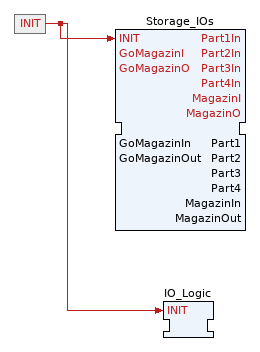
      [picture p72: application VDMA_Station1_EmulatorApp_SingleDevice.Storage]
      SUBAPPLICATION Storage_IOs
        EVENT_INPUT
          INIT;
          GoMagazinI;
          GoMagazinO;
        END_EVENT
        EVENT_OUTPUT
          Part1In;
          Part2In;
          Part3In;
          Part4In;
          MagazinI;
          MagazinO;
        END_EVENT
        VAR_INPUT
          GoMagazinIn : BOOL;
          GoMagazinOut : BOOL;
        END_VAR
        VAR_OUTPUT
          Part1 : BOOL;
          Part2 : BOOL;
          Part3 : BOOL;
          Part4 : BOOL;
          MagazinIn : BOOL;
          MagazinOut : BOOL;
        END_VAR
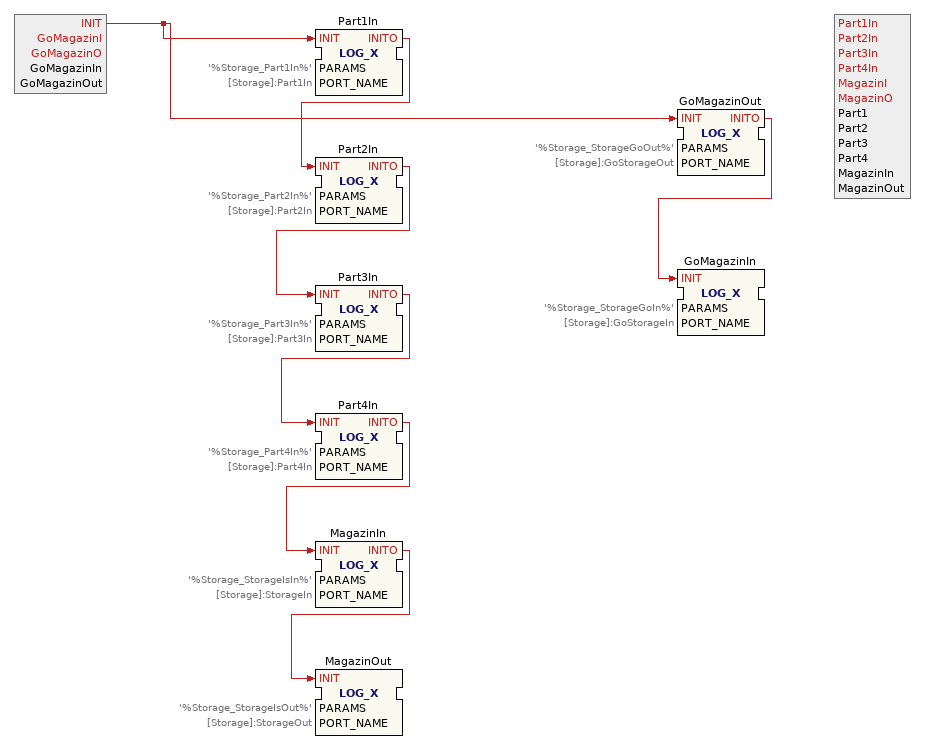
        FBS
          GoMagazinIn : LOG_X(PARAMS := '%Storage_StorageGoIn%', PORT_NAME := [Storage]:GoStorageIn);
          GoMagazinOut : LOG_X(PARAMS := '%Storage_StorageGoOut%', PORT_NAME := [Storage]:GoStorageOut);
          MagazinOut : LOG_X(PARAMS := '%Storage_StorageIsOut%', PORT_NAME := [Storage]:StorageOut);
          MagazinIn : LOG_X(PARAMS := '%Storage_StorageIsIn%', PORT_NAME := [Storage]:StorageIn);
          Part4In : LOG_X(PARAMS := '%Storage_Part4In%', PORT_NAME := [Storage]:Part4In);
          Part3In : LOG_X(PARAMS := '%Storage_Part3In%', PORT_NAME := [Storage]:Part3In);
          Part2In : LOG_X(PARAMS := '%Storage_Part2In%', PORT_NAME := [Storage]:Part2In);
          Part1In : LOG_X(PARAMS := '%Storage_Part1In%', PORT_NAME := [Storage]:Part1In);
        END_FBS
        EVENT_CONNECTIONS
          GoMagazinOut.INITO TO GoMagazinIn.INIT;
          MagazinIn.INITO TO MagazinOut.INIT;
          Part4In.INITO TO MagazinIn.INIT;
          Part3In.INITO TO Part4In.INIT;
          Part2In.INITO TO Part3In.INIT;
          Part1In.INITO TO Part2In.INIT;
          INIT TO Part1In.INIT;
          INIT TO GoMagazinOut.INIT;
        END_CONNECTIONS
      END_SUBAPPLICATION
      SUBAPPLICATION IO_Logic
        EVENT_INPUT
          INIT;
        END_EVENT
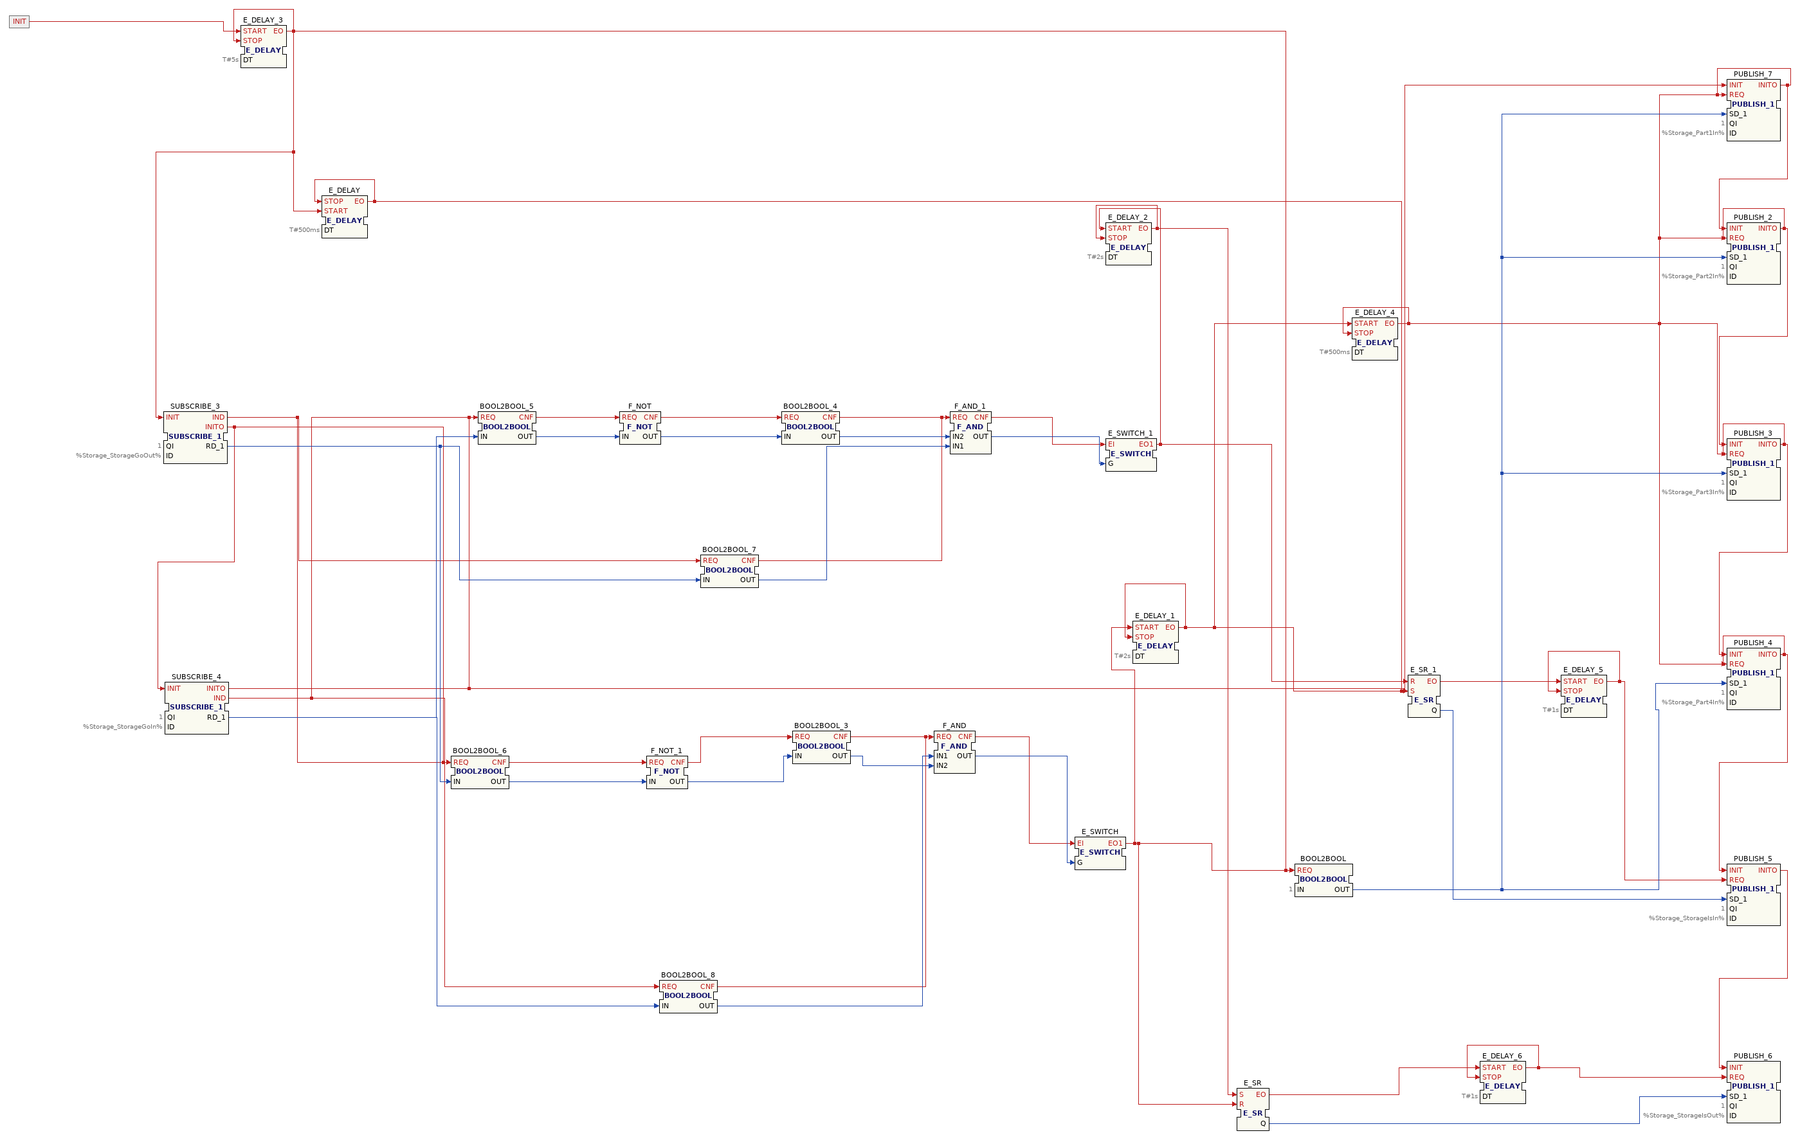
        FBS
          E_SWITCH_1 : E_SWITCH;
          BOOL2BOOL_4 : BOOL2BOOL;
          F_NOT : F_NOT;
          PUBLISH_3 : PUBLISH_1(QI := 1, ID := %Storage_Part3In%);
          BOOL2BOOL_6 : BOOL2BOOL;
          E_SR_1 : E_SR;
          F_NOT_1 : F_NOT;
          PUBLISH_7 : PUBLISH_1(QI := 1, ID := %Storage_Part1In%);
          BOOL2BOOL : BOOL2BOOL(IN := 1);
          BOOL2BOOL_5 : BOOL2BOOL;
          BOOL2BOOL_7 : BOOL2BOOL;
          E_SR : E_SR;
          F_AND_1 : F_AND;
          SUBSCRIBE_4 : SUBSCRIBE_1(QI := 1, ID := %Storage_StorageGoIn%);
          SUBSCRIBE_3 : SUBSCRIBE_1(QI := 1, ID := %Storage_StorageGoOut%);
          PUBLISH_6 : PUBLISH_1(QI := 1, ID := %Storage_StorageIsOut%);
          F_AND : F_AND;
          BOOL2BOOL_3 : BOOL2BOOL;
          PUBLISH_5 : PUBLISH_1(QI := 1, ID := %Storage_StorageIsIn%);
          PUBLISH_4 : PUBLISH_1(QI := 1, ID := %Storage_Part4In%);
          E_DELAY_2 : E_DELAY(DT := T#2s);
          BOOL2BOOL_8 : BOOL2BOOL;
          E_DELAY_1 : E_DELAY(DT := T#2s);
          PUBLISH_2 : PUBLISH_1(QI := 1, ID := %Storage_Part2In%);
          E_SWITCH : E_SWITCH;
          E_DELAY : E_DELAY(DT := T#500ms);
          E_DELAY_3 : E_DELAY(DT := T#5s);
          E_DELAY_4 : E_DELAY(DT := T#500ms);
          E_DELAY_5 : E_DELAY(DT := T#1s);
          E_DELAY_6 : E_DELAY(DT := T#1s);
        END_FBS
        EVENT_CONNECTIONS
          F_AND_1.CNF TO E_SWITCH_1.EI;
          E_SWITCH_1.EO1 TO E_SR_1.R;
          E_SWITCH_1.EO1 TO E_DELAY_2.START;
          F_NOT.CNF TO BOOL2BOOL_4.REQ;
          BOOL2BOOL_4.CNF TO F_AND_1.REQ;
          BOOL2BOOL_5.CNF TO F_NOT.REQ;
          PUBLISH_2.INITO TO PUBLISH_3.INIT;
          PUBLISH_3.INITO TO PUBLISH_3.REQ;
          PUBLISH_3.INITO TO PUBLISH_4.INIT;
          SUBSCRIBE_3.IND TO BOOL2BOOL_6.REQ;
          SUBSCRIBE_3.INITO TO BOOL2BOOL_6.REQ;
          BOOL2BOOL_6.CNF TO F_NOT_1.REQ;
          E_DELAY_1.EO TO E_SR_1.S;
          F_NOT_1.CNF TO BOOL2BOOL_3.REQ;
          SUBSCRIBE_4.INITO TO PUBLISH_7.INIT;
          PUBLISH_7.INITO TO PUBLISH_7.REQ;
          PUBLISH_7.INITO TO PUBLISH_2.INIT;
          E_SWITCH.EO1 TO BOOL2BOOL.REQ;
          SUBSCRIBE_4.IND TO BOOL2BOOL_5.REQ;
          SUBSCRIBE_4.INITO TO BOOL2BOOL_5.REQ;
          SUBSCRIBE_3.IND TO BOOL2BOOL_7.REQ;
          BOOL2BOOL_7.CNF TO F_AND_1.REQ;
          E_DELAY_2.EO TO E_SR.S;
          E_SWITCH.EO1 TO E_SR.R;
          SUBSCRIBE_3.INITO TO SUBSCRIBE_4.INIT;
          SUBSCRIBE_4.IND TO BOOL2BOOL_8.REQ;
          PUBLISH_5.INITO TO PUBLISH_6.INIT;
          BOOL2BOOL_3.CNF TO F_AND.REQ;
          BOOL2BOOL_8.CNF TO F_AND.REQ;
          F_AND.CNF TO E_SWITCH.EI;
          PUBLISH_4.INITO TO PUBLISH_5.INIT;
          PUBLISH_4.INITO TO PUBLISH_4.REQ;
          E_DELAY_2.EO TO E_DELAY_2.STOP;
          E_SWITCH.EO1 TO E_DELAY_1.START;
          E_DELAY_1.EO TO E_DELAY_1.STOP;
          PUBLISH_2.INITO TO PUBLISH_2.REQ;
          E_DELAY.EO TO E_DELAY.STOP;
          E_DELAY.EO TO E_SR_1.S;
          E_DELAY_3.EO TO BOOL2BOOL.REQ;
          E_DELAY_3.EO TO E_DELAY.START;
          E_DELAY_3.EO TO SUBSCRIBE_3.INIT;
          INIT TO E_DELAY_3.START;
          E_DELAY_3.EO TO E_DELAY_3.STOP;
          E_DELAY_4.EO TO PUBLISH_2.REQ;
          E_DELAY_4.EO TO PUBLISH_4.REQ;
          E_DELAY_4.EO TO PUBLISH_7.REQ;
          E_DELAY_4.EO TO PUBLISH_3.REQ;
          E_DELAY_1.EO TO E_DELAY_4.START;
          E_DELAY_4.EO TO E_DELAY_4.STOP;
          E_SR_1.EO TO E_DELAY_5.START;
          E_DELAY_5.EO TO PUBLISH_5.REQ;
          E_DELAY_5.EO TO E_DELAY_5.STOP;
          E_SR.EO TO E_DELAY_6.START;
          E_DELAY_6.EO TO PUBLISH_6.REQ;
          E_DELAY_6.EO TO E_DELAY_6.STOP;
        END_CONNECTIONS
        DATA_CONNECTIONS
          F_AND_1.OUT TO E_SWITCH_1.G;
          F_NOT.OUT TO BOOL2BOOL_4.IN;
          BOOL2BOOL_4.OUT TO F_AND_1.IN2;
          BOOL2BOOL_5.OUT TO F_NOT.IN;
          BOOL2BOOL.OUT TO PUBLISH_3.SD_1;
          SUBSCRIBE_3.RD_1 TO BOOL2BOOL_6.IN;
          BOOL2BOOL_6.OUT TO F_NOT_1.IN;
          F_NOT_1.OUT TO BOOL2BOOL_3.IN;
          BOOL2BOOL.OUT TO PUBLISH_7.SD_1;
          BOOL2BOOL.OUT TO PUBLISH_4.SD_1;
          BOOL2BOOL.OUT TO PUBLISH_2.SD_1;
          SUBSCRIBE_4.RD_1 TO BOOL2BOOL_5.IN;
          SUBSCRIBE_3.RD_1 TO BOOL2BOOL_7.IN;
          BOOL2BOOL_7.OUT TO F_AND_1.IN1;
          E_SR.Q TO PUBLISH_6.SD_1;
          SUBSCRIBE_4.RD_1 TO BOOL2BOOL_8.IN;
          BOOL2BOOL_8.OUT TO F_AND.IN1;
          BOOL2BOOL_3.OUT TO F_AND.IN2;
          F_AND.OUT TO E_SWITCH.G;
          E_SR_1.Q TO PUBLISH_5.SD_1;
        END_CONNECTIONS
      END_SUBAPPLICATION
      EVENT_CONNECTIONS
        INIT TO Storage_IOs.INIT;
        INIT TO IO_Logic.INIT;
      END_CONNECTIONS
    END_SUBAPPLICATION
    SUBAPPLICATION Gripper1
      EVENT_INPUT
        INIT;
      END_EVENT
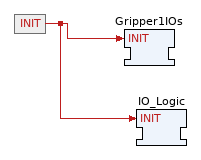
      SUBAPPLICATION Gripper1IOs
        EVENT_INPUT
          INIT;
        END_EVENT
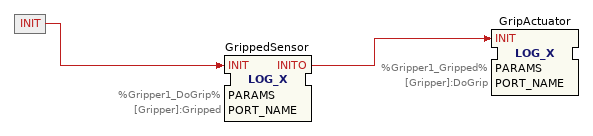
        FBS
          GripActuator : LOG_X(PARAMS := %Gripper1_Gripped%, PORT_NAME := [Gripper]:DoGrip);
          GrippedSensor : LOG_X(PARAMS := %Gripper1_DoGrip%, PORT_NAME := [Gripper]:Gripped);
        END_FBS
        EVENT_CONNECTIONS
          INIT TO GrippedSensor.INIT;
          GrippedSensor.INITO TO GripActuator.INIT;
        END_CONNECTIONS
      END_SUBAPPLICATION
      SUBAPPLICATION IO_Logic
        EVENT_INPUT
          INIT;
        END_EVENT
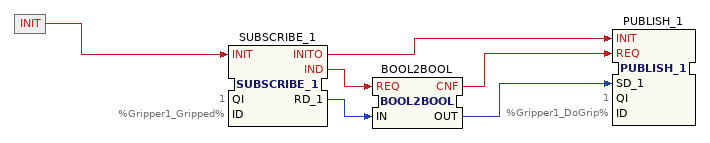
        FBS
          SUBSCRIBE_1 : SUBSCRIBE_1(QI := 1, ID := %Gripper1_Gripped%);
          BOOL2BOOL : BOOL2BOOL;
          PUBLISH_1 : PUBLISH_1(QI := 1, ID := %Gripper1_DoGrip%);
        END_FBS
        EVENT_CONNECTIONS
          SUBSCRIBE_1.INITO TO PUBLISH_1.INIT;
          SUBSCRIBE_1.IND TO BOOL2BOOL.REQ;
          BOOL2BOOL.CNF TO PUBLISH_1.REQ;
          INIT TO SUBSCRIBE_1.INIT;
        END_CONNECTIONS
        DATA_CONNECTIONS
          SUBSCRIBE_1.RD_1 TO BOOL2BOOL.IN;
          BOOL2BOOL.OUT TO PUBLISH_1.SD_1;
        END_CONNECTIONS
      END_SUBAPPLICATION
      EVENT_CONNECTIONS
        INIT TO IO_Logic.INIT;
        INIT TO Gripper1IOs.INIT;
      END_CONNECTIONS
    END_SUBAPPLICATION
    SUBAPPLICATION Gripper2
      EVENT_INPUT
        INIT;
      END_EVENT
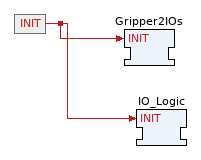
      SUBAPPLICATION Gripper2IOs
        EVENT_INPUT
          INIT;
        END_EVENT
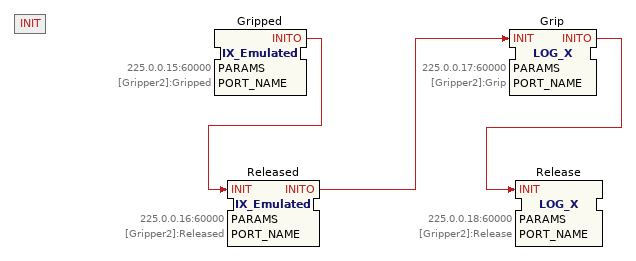
        FBS
          Grip : LOG_X(PARAMS := 225.0.0.17:60000, PORT_NAME := [Gripper2]:Grip);
          Gripped : IX_Emulated(PARAMS := 225.0.0.15:60000, PORT_NAME := [Gripper2]:Gripped);
          Released : IX_Emulated(PARAMS := 225.0.0.16:60000, PORT_NAME := [Gripper2]:Released);
          Release : LOG_X(PARAMS := 225.0.0.18:60000, PORT_NAME := [Gripper2]:Release);
        END_FBS
        EVENT_CONNECTIONS
          Gripped.INITO TO Released.INIT;
          Released.INITO TO Grip.INIT;
          Grip.INITO TO Release.INIT;
        END_CONNECTIONS
      END_SUBAPPLICATION
      SUBAPPLICATION IO_Logic
        EVENT_INPUT
          INIT;
        END_EVENT
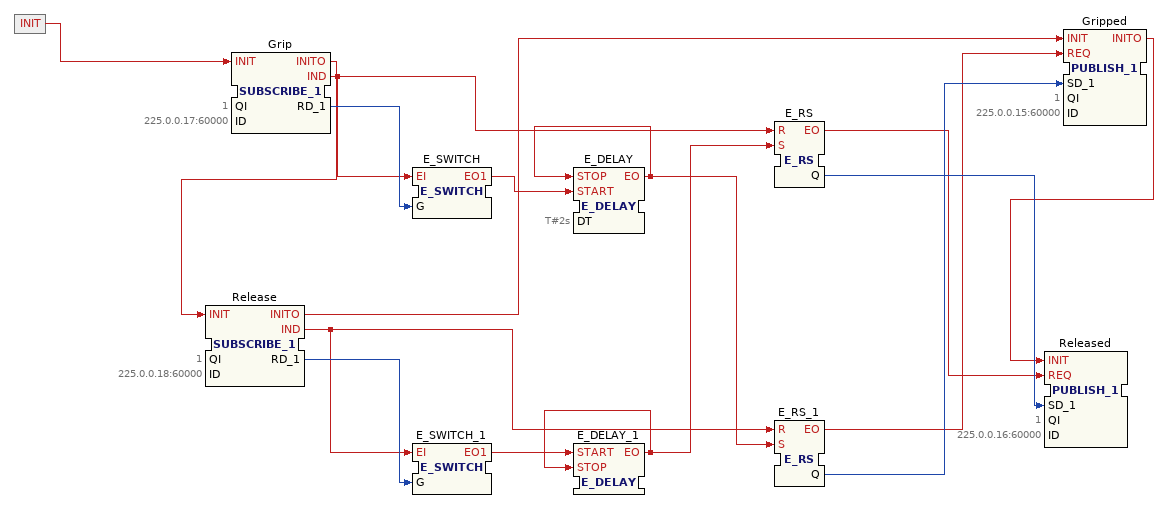
        FBS
          Grip : SUBSCRIBE_1(QI := 1, ID := 225.0.0.17:60000);
          Gripped : PUBLISH_1(QI := 1, ID := 225.0.0.15:60000);
          Release : SUBSCRIBE_1(QI := 1, ID := 225.0.0.18:60000);
          Released : PUBLISH_1(QI := 1, ID := 225.0.0.16:60000);
          E_DELAY : E_DELAY(DT := T#2s);
          E_RS : E_RS;
          E_RS_1 : E_RS;
          E_DELAY_1 : E_DELAY;
          E_SWITCH : E_SWITCH;
          E_SWITCH_1 : E_SWITCH;
        END_FBS
        EVENT_CONNECTIONS
          INIT TO Grip.INIT;
          Grip.INITO TO Release.INIT;
          Release.INITO TO Gripped.INIT;
          Gripped.INITO TO Released.INIT;
          E_DELAY.EO TO E_DELAY.STOP;
          Grip.IND TO E_RS.R;
          E_RS.EO TO Released.REQ;
          Release.IND TO E_RS_1.R;
          E_RS_1.EO TO Gripped.REQ;
          E_DELAY.EO TO E_RS_1.S;
          Grip.IND TO E_SWITCH.EI;
          E_SWITCH.EO1 TO E_DELAY.START;
          Release.IND TO E_SWITCH_1.EI;
          E_SWITCH_1.EO1 TO E_DELAY_1.START;
          E_DELAY_1.EO TO E_DELAY_1.STOP;
          E_DELAY_1.EO TO E_RS.S;
        END_CONNECTIONS
        DATA_CONNECTIONS
          E_RS.Q TO Released.SD_1;
          E_RS_1.Q TO Gripped.SD_1;
          Grip.RD_1 TO E_SWITCH.G;
          Release.RD_1 TO E_SWITCH_1.G;
        END_CONNECTIONS
      END_SUBAPPLICATION
      EVENT_CONNECTIONS
        INIT TO Gripper2IOs.INIT;
        INIT TO IO_Logic.INIT;
      END_CONNECTIONS
    END_SUBAPPLICATION
    SUBAPPLICATION IOs_to_OPCUA
      EVENT_INPUT
        INIT;
      END_EVENT
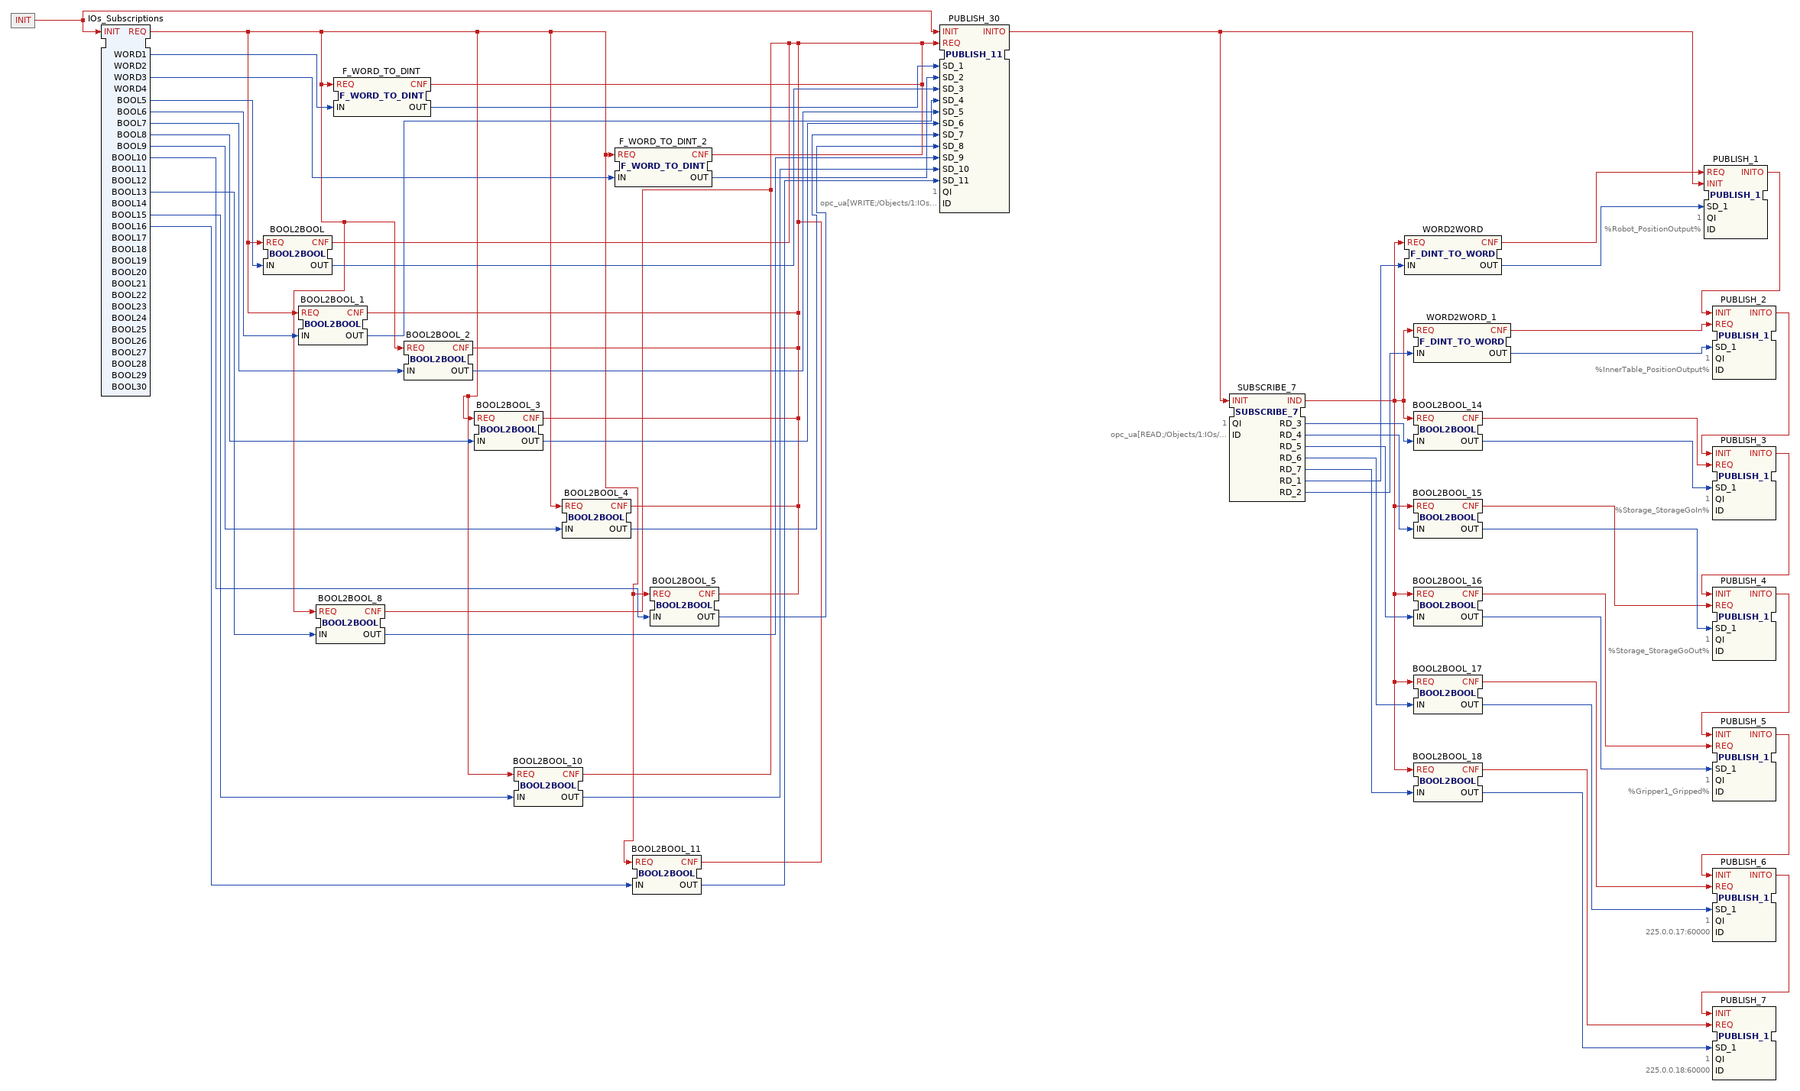
      FBS
        F_WORD_TO_DINT : F_WORD_TO_DINT;
        F_WORD_TO_DINT_2 : F_WORD_TO_DINT;
        BOOL2BOOL : BOOL2BOOL;
        BOOL2BOOL_1 : BOOL2BOOL;
        BOOL2BOOL_2 : BOOL2BOOL;
        BOOL2BOOL_3 : BOOL2BOOL;
        BOOL2BOOL_4 : BOOL2BOOL;
        BOOL2BOOL_5 : BOOL2BOOL;
        BOOL2BOOL_8 : BOOL2BOOL;
        BOOL2BOOL_10 : BOOL2BOOL;
        BOOL2BOOL_11 : BOOL2BOOL;
        SUBSCRIBE_7 : SUBSCRIBE_7(QI := 1, ID := opc_ua[READ;/Objects/1:IOs/1:Robot.PresetPosition;/Objects/1:IOs/1:InnerTable.PresetPosition;/Objects/1:IOs/1:Storage.GoMagazinIn;/Objects/1:IOs/1:Storage.GoMagazinOut;/Objects/1:IOs/1:Gripper1.Grip;/Objects/1:IOs/1:Gripper2.Grip;/Objects/1:IOs/1:Gripper2.Release]);
        BOOL2BOOL_14 : BOOL2BOOL;
        BOOL2BOOL_15 : BOOL2BOOL;
        BOOL2BOOL_16 : BOOL2BOOL;
        BOOL2BOOL_17 : BOOL2BOOL;
        BOOL2BOOL_18 : BOOL2BOOL;
        WORD2WORD : F_DINT_TO_WORD;
        WORD2WORD_1 : F_DINT_TO_WORD;
        PUBLISH_1 : PUBLISH_1(QI := 1, ID := %Robot_PositionOutput%);
        PUBLISH_2 : PUBLISH_1(QI := 1, ID := %InnerTable_PositionOutput%);
        PUBLISH_3 : PUBLISH_1(QI := 1, ID := %Storage_StorageGoIn%);
        PUBLISH_4 : PUBLISH_1(QI := 1, ID := %Storage_StorageGoOut%);
        PUBLISH_5 : PUBLISH_1(QI := 1, ID := %Gripper1_Gripped%);
        PUBLISH_6 : PUBLISH_1(QI := 1, ID := 225.0.0.17:60000);
        PUBLISH_7 : PUBLISH_1(QI := 1, ID := 225.0.0.18:60000);
        PUBLISH_30 : PUBLISH_11(QI := 1, ID := opc_ua[WRITE;/Objects/1:IOs/1:Robot.CurrentPosition;/Objects/1:IOs/1:InnerTable.CurrentPosition;/Objects/1:IOs/1:Storage.Part1In;/Objects/1:IOs/1:Storage.Part2In;/Objects/1:IOs/1:Storage.Part3In;/Objects/1:IOs/1:Storage.Part4In;/Objects/1:IOs/1:Storage.MagazinIn;/Objects/1:IOs/1:Storage.MagazinOut;/Objects/1:IOs/1:Gripper1.Gripped;/Objects/1:IOs/1:Gripper2.Gripped;/Objects/1:IOs/1:Gripper2.Released]);
      END_FBS
      SUBAPPLICATION IOs_Subscriptions
        EVENT_INPUT
          INIT;
        END_EVENT
        EVENT_OUTPUT
          REQ;
        END_EVENT
        VAR_OUTPUT
          WORD1 : WORD;
          WORD2 : WORD;
          WORD3 : WORD;
          WORD4 : WORD;
          BOOL5 : BOOL;
          BOOL6 : BOOL;
          BOOL7 : BOOL;
          BOOL8 : BOOL;
          BOOL9 : BOOL;
          BOOL10 : BOOL;
          BOOL11 : BOOL;
          BOOL12 : BOOL;
          BOOL13 : BOOL;
          BOOL14 : BOOL;
          BOOL15 : BOOL;
          BOOL16 : BOOL;
          BOOL17 : BOOL;
          BOOL18 : BOOL;
          BOOL19 : BOOL;
          BOOL20 : BOOL;
          BOOL21 : BOOL;
          BOOL22 : BOOL;
          BOOL23 : BOOL;
          BOOL24 : BOOL;
          BOOL25 : BOOL;
          BOOL26 : BOOL;
          BOOL27 : BOOL;
          BOOL28 : BOOL;
          BOOL29 : BOOL;
          BOOL30 : BOOL;
        END_VAR
        FBS
          SUBSCRIBE_1 : SUBSCRIBE_1(QI := 1, ID := %Robot_PositionInput%);
          SUBSCRIBE_2 : SUBSCRIBE_1(QI := 1, ID := %Robot_PositionOutput%);
          SUBSCRIBE_3 : SUBSCRIBE_1(QI := 1, ID := %InnerTable_PositionInput%);
          SUBSCRIBE_4 : SUBSCRIBE_1(QI := 1, ID := %InnerTable_PositionOutput%);
          SUBSCRIBE_5 : SUBSCRIBE_1(QI := 1, ID := %Storage_Part1In%);
          SUBSCRIBE_6 : SUBSCRIBE_1(QI := 1, ID := %Storage_Part2In%);
          SUBSCRIBE_7 : SUBSCRIBE_1(QI := 1, ID := %Storage_Part3In%);
          SUBSCRIBE_8 : SUBSCRIBE_1(QI := 1, ID := %Storage_Part4In%);
          SUBSCRIBE_9 : SUBSCRIBE_1(QI := 1, ID := %Storage_StorageIsIn%);
          SUBSCRIBE_10 : SUBSCRIBE_1(QI := 1, ID := %Storage_StorageIsOut%);
          SUBSCRIBE_11 : SUBSCRIBE_1(QI := 1, ID := %Storage_StorageGoOut%);
          SUBSCRIBE_12 : SUBSCRIBE_1(QI := 1, ID := %Storage_StorageGoIn%);
          SUBSCRIBE_13 : SUBSCRIBE_1(QI := 1, ID := %Gripper1_DoGrip%);
          SUBSCRIBE_14 : SUBSCRIBE_1(QI := 1, ID := %Gripper1_Gripped%);
          SUBSCRIBE_15 : SUBSCRIBE_1(QI := 1, ID := 225.0.0.15:60000);
          SUBSCRIBE_16 : SUBSCRIBE_1(QI := 1, ID := 225.0.0.16:60000);
          SUBSCRIBE_17 : SUBSCRIBE_1(QI := 1, ID := 225.0.0.17:60000);
          SUBSCRIBE_18 : SUBSCRIBE_1(QI := 1, ID := 225.0.0.18:60000);
          SUBSCRIBE_19 : SUBSCRIBE_1;
          SUBSCRIBE_20 : SUBSCRIBE_1;
          SUBSCRIBE_21 : SUBSCRIBE_1;
          SUBSCRIBE_22 : SUBSCRIBE_1;
          SUBSCRIBE_23 : SUBSCRIBE_1;
          SUBSCRIBE_24 : SUBSCRIBE_1;
          SUBSCRIBE_25 : SUBSCRIBE_1;
          SUBSCRIBE_26 : SUBSCRIBE_1;
          SUBSCRIBE_27 : SUBSCRIBE_1;
          SUBSCRIBE_28 : SUBSCRIBE_1;
          SUBSCRIBE_29 : SUBSCRIBE_1;
          SUBSCRIBE_30 : SUBSCRIBE_1;
        END_FBS
        EVENT_CONNECTIONS
          SUBSCRIBE_1.IND TO REQ;
          SUBSCRIBE_2.IND TO REQ;
          SUBSCRIBE_3.IND TO REQ;
          SUBSCRIBE_4.IND TO REQ;
          SUBSCRIBE_5.IND TO REQ;
          SUBSCRIBE_6.IND TO REQ;
          SUBSCRIBE_7.IND TO REQ;
          SUBSCRIBE_8.IND TO REQ;
          SUBSCRIBE_9.IND TO REQ;
          SUBSCRIBE_10.IND TO REQ;
          SUBSCRIBE_11.IND TO REQ;
          SUBSCRIBE_12.IND TO REQ;
          SUBSCRIBE_13.IND TO REQ;
          SUBSCRIBE_14.IND TO REQ;
          SUBSCRIBE_15.IND TO REQ;
          SUBSCRIBE_16.IND TO REQ;
          SUBSCRIBE_17.IND TO REQ;
          SUBSCRIBE_18.IND TO REQ;
          SUBSCRIBE_19.IND TO REQ;
          SUBSCRIBE_20.IND TO REQ;
          SUBSCRIBE_21.IND TO REQ;
          SUBSCRIBE_22.IND TO REQ;
          SUBSCRIBE_23.IND TO REQ;
          SUBSCRIBE_24.IND TO REQ;
          SUBSCRIBE_25.IND TO REQ;
          SUBSCRIBE_26.IND TO REQ;
          SUBSCRIBE_27.IND TO REQ;
          SUBSCRIBE_28.IND TO REQ;
          SUBSCRIBE_29.IND TO REQ;
          SUBSCRIBE_30.IND TO REQ;
          SUBSCRIBE_1.INITO TO SUBSCRIBE_2.INIT;
          SUBSCRIBE_2.INITO TO SUBSCRIBE_3.INIT;
          SUBSCRIBE_3.INITO TO SUBSCRIBE_4.INIT;
          SUBSCRIBE_4.INITO TO SUBSCRIBE_5.INIT;
          SUBSCRIBE_5.INITO TO SUBSCRIBE_6.INIT;
          SUBSCRIBE_6.INITO TO SUBSCRIBE_7.INIT;
          SUBSCRIBE_7.INITO TO SUBSCRIBE_8.INIT;
          SUBSCRIBE_8.INITO TO SUBSCRIBE_9.INIT;
          SUBSCRIBE_9.INITO TO SUBSCRIBE_10.INIT;
          SUBSCRIBE_10.INITO TO SUBSCRIBE_11.INIT;
          SUBSCRIBE_11.INITO TO SUBSCRIBE_12.INIT;
          SUBSCRIBE_12.INITO TO SUBSCRIBE_13.INIT;
          SUBSCRIBE_13.INITO TO SUBSCRIBE_14.INIT;
          SUBSCRIBE_14.INITO TO SUBSCRIBE_15.INIT;
          SUBSCRIBE_15.INITO TO SUBSCRIBE_16.INIT;
          SUBSCRIBE_16.INITO TO SUBSCRIBE_17.INIT;
          SUBSCRIBE_17.INITO TO SUBSCRIBE_18.INIT;
          SUBSCRIBE_18.INITO TO SUBSCRIBE_19.INIT;
          SUBSCRIBE_19.INITO TO SUBSCRIBE_20.INIT;
          SUBSCRIBE_20.INITO TO SUBSCRIBE_21.INIT;
          SUBSCRIBE_21.INITO TO SUBSCRIBE_22.INIT;
          SUBSCRIBE_22.INITO TO SUBSCRIBE_23.INIT;
          SUBSCRIBE_23.INITO TO SUBSCRIBE_24.INIT;
          SUBSCRIBE_24.INITO TO SUBSCRIBE_25.INIT;
          SUBSCRIBE_25.INITO TO SUBSCRIBE_26.INIT;
          SUBSCRIBE_26.INITO TO SUBSCRIBE_27.INIT;
          SUBSCRIBE_27.INITO TO SUBSCRIBE_28.INIT;
          SUBSCRIBE_28.INITO TO SUBSCRIBE_29.INIT;
          SUBSCRIBE_29.INITO TO SUBSCRIBE_30.INIT;
          INIT TO SUBSCRIBE_1.INIT;
        END_CONNECTIONS
        DATA_CONNECTIONS
          SUBSCRIBE_30.RD_1 TO BOOL30;
          SUBSCRIBE_29.RD_1 TO BOOL29;
          SUBSCRIBE_28.RD_1 TO BOOL28;
          SUBSCRIBE_27.RD_1 TO BOOL27;
          SUBSCRIBE_26.RD_1 TO BOOL26;
          SUBSCRIBE_25.RD_1 TO BOOL25;
          SUBSCRIBE_24.RD_1 TO BOOL24;
          SUBSCRIBE_23.RD_1 TO BOOL23;
          SUBSCRIBE_22.RD_1 TO BOOL22;
          SUBSCRIBE_21.RD_1 TO BOOL21;
          SUBSCRIBE_20.RD_1 TO BOOL20;
          SUBSCRIBE_19.RD_1 TO BOOL19;
          SUBSCRIBE_18.RD_1 TO BOOL18;
          SUBSCRIBE_17.RD_1 TO BOOL17;
          SUBSCRIBE_16.RD_1 TO BOOL16;
          SUBSCRIBE_15.RD_1 TO BOOL15;
          SUBSCRIBE_14.RD_1 TO BOOL14;
          SUBSCRIBE_13.RD_1 TO BOOL13;
          SUBSCRIBE_12.RD_1 TO BOOL12;
          SUBSCRIBE_11.RD_1 TO BOOL11;
          SUBSCRIBE_10.RD_1 TO BOOL10;
          SUBSCRIBE_9.RD_1 TO BOOL9;
          SUBSCRIBE_8.RD_1 TO BOOL8;
          SUBSCRIBE_7.RD_1 TO BOOL7;
          SUBSCRIBE_6.RD_1 TO BOOL6;
          SUBSCRIBE_5.RD_1 TO BOOL5;
          SUBSCRIBE_1.RD_1 TO WORD1;
          SUBSCRIBE_2.RD_1 TO WORD2;
          SUBSCRIBE_3.RD_1 TO WORD3;
          SUBSCRIBE_4.RD_1 TO WORD4;
        END_CONNECTIONS
      END_SUBAPPLICATION
      EVENT_CONNECTIONS
        INIT TO IOs_Subscriptions.INIT;
        IOs_Subscriptions.REQ TO F_WORD_TO_DINT.REQ;
        IOs_Subscriptions.REQ TO F_WORD_TO_DINT_2.REQ;
        IOs_Subscriptions.REQ TO BOOL2BOOL.REQ;
        IOs_Subscriptions.REQ TO BOOL2BOOL_1.REQ;
        IOs_Subscriptions.REQ TO BOOL2BOOL_2.REQ;
        IOs_Subscriptions.REQ TO BOOL2BOOL_3.REQ;
        IOs_Subscriptions.REQ TO BOOL2BOOL_4.REQ;
        IOs_Subscriptions.REQ TO BOOL2BOOL_5.REQ;
        IOs_Subscriptions.REQ TO BOOL2BOOL_8.REQ;
        IOs_Subscriptions.REQ TO BOOL2BOOL_10.REQ;
        IOs_Subscriptions.REQ TO BOOL2BOOL_11.REQ;
        SUBSCRIBE_7.IND TO BOOL2BOOL_14.REQ;
        SUBSCRIBE_7.IND TO BOOL2BOOL_15.REQ;
        SUBSCRIBE_7.IND TO BOOL2BOOL_16.REQ;
        SUBSCRIBE_7.IND TO BOOL2BOOL_17.REQ;
        SUBSCRIBE_7.IND TO BOOL2BOOL_18.REQ;
        SUBSCRIBE_7.IND TO WORD2WORD.REQ;
        SUBSCRIBE_7.IND TO WORD2WORD_1.REQ;
        PUBLISH_1.INITO TO PUBLISH_2.INIT;
        PUBLISH_2.INITO TO PUBLISH_3.INIT;
        PUBLISH_3.INITO TO PUBLISH_4.INIT;
        PUBLISH_4.INITO TO PUBLISH_5.INIT;
        PUBLISH_5.INITO TO PUBLISH_6.INIT;
        WORD2WORD.CNF TO PUBLISH_1.REQ;
        WORD2WORD_1.CNF TO PUBLISH_2.REQ;
        BOOL2BOOL_14.CNF TO PUBLISH_3.REQ;
        BOOL2BOOL_15.CNF TO PUBLISH_4.REQ;
        BOOL2BOOL_16.CNF TO PUBLISH_5.REQ;
        BOOL2BOOL_17.CNF TO PUBLISH_6.REQ;
        PUBLISH_6.INITO TO PUBLISH_7.INIT;
        BOOL2BOOL_18.CNF TO PUBLISH_7.REQ;
        INIT TO PUBLISH_30.INIT;
        F_WORD_TO_DINT.CNF TO PUBLISH_30.REQ;
        F_WORD_TO_DINT_2.CNF TO PUBLISH_30.REQ;
        BOOL2BOOL.CNF TO PUBLISH_30.REQ;
        BOOL2BOOL_1.CNF TO PUBLISH_30.REQ;
        BOOL2BOOL_2.CNF TO PUBLISH_30.REQ;
        BOOL2BOOL_3.CNF TO PUBLISH_30.REQ;
        BOOL2BOOL_4.CNF TO PUBLISH_30.REQ;
        BOOL2BOOL_5.CNF TO PUBLISH_30.REQ;
        BOOL2BOOL_8.CNF TO PUBLISH_30.REQ;
        BOOL2BOOL_10.CNF TO PUBLISH_30.REQ;
        BOOL2BOOL_11.CNF TO PUBLISH_30.REQ;
        PUBLISH_30.INITO TO SUBSCRIBE_7.INIT;
        PUBLISH_30.INITO TO PUBLISH_1.INIT;
      END_CONNECTIONS
      DATA_CONNECTIONS
        IOs_Subscriptions.WORD1 TO F_WORD_TO_DINT.IN;
        IOs_Subscriptions.WORD3 TO F_WORD_TO_DINT_2.IN;
        IOs_Subscriptions.BOOL5 TO BOOL2BOOL.IN;
        IOs_Subscriptions.BOOL6 TO BOOL2BOOL_1.IN;
        IOs_Subscriptions.BOOL7 TO BOOL2BOOL_2.IN;
        IOs_Subscriptions.BOOL8 TO BOOL2BOOL_3.IN;
        IOs_Subscriptions.BOOL9 TO BOOL2BOOL_4.IN;
        IOs_Subscriptions.BOOL10 TO BOOL2BOOL_5.IN;
        IOs_Subscriptions.BOOL13 TO BOOL2BOOL_8.IN;
        IOs_Subscriptions.BOOL15 TO BOOL2BOOL_10.IN;
        IOs_Subscriptions.BOOL16 TO BOOL2BOOL_11.IN;
        SUBSCRIBE_7.RD_3 TO BOOL2BOOL_14.IN;
        SUBSCRIBE_7.RD_4 TO BOOL2BOOL_15.IN;
        SUBSCRIBE_7.RD_5 TO BOOL2BOOL_16.IN;
        SUBSCRIBE_7.RD_6 TO BOOL2BOOL_17.IN;
        SUBSCRIBE_7.RD_7 TO BOOL2BOOL_18.IN;
        SUBSCRIBE_7.RD_1 TO WORD2WORD.IN;
        SUBSCRIBE_7.RD_2 TO WORD2WORD_1.IN;
        WORD2WORD.OUT TO PUBLISH_1.SD_1;
        WORD2WORD_1.OUT TO PUBLISH_2.SD_1;
        BOOL2BOOL_14.OUT TO PUBLISH_3.SD_1;
        BOOL2BOOL_15.OUT TO PUBLISH_4.SD_1;
        BOOL2BOOL_16.OUT TO PUBLISH_5.SD_1;
        BOOL2BOOL_17.OUT TO PUBLISH_6.SD_1;
        BOOL2BOOL_18.OUT TO PUBLISH_7.SD_1;
        F_WORD_TO_DINT.OUT TO PUBLISH_30.SD_1;
        F_WORD_TO_DINT_2.OUT TO PUBLISH_30.SD_2;
        BOOL2BOOL.OUT TO PUBLISH_30.SD_3;
        BOOL2BOOL_1.OUT TO PUBLISH_30.SD_4;
        BOOL2BOOL_2.OUT TO PUBLISH_30.SD_5;
        BOOL2BOOL_3.OUT TO PUBLISH_30.SD_6;
        BOOL2BOOL_4.OUT TO PUBLISH_30.SD_7;
        BOOL2BOOL_5.OUT TO PUBLISH_30.SD_8;
        BOOL2BOOL_8.OUT TO PUBLISH_30.SD_9;
        BOOL2BOOL_10.OUT TO PUBLISH_30.SD_10;
        BOOL2BOOL_11.OUT TO PUBLISH_30.SD_11;
      END_CONNECTIONS
    END_SUBAPPLICATION
  END_APPLICATION
  APPLICATION VDMA_Station1_HierarchicalControl_Distributed_SingleDevice
    FBS
      SERVER_2 : SERVER_0_1(QI := 1, ID := opc_ua[CREATE_METHOD;/Objects/Robot/PresetPositionUpd]);
      PUBLISH_3 : PUBLISH_1(QI := 1, ID := opc_ua[WRITE;/Objects/Turntable/CurrentPosition]);
      SERVER_0 : SERVER_0(QI := 1, ID := opc_ua[CREATE_METHOD;/Objects/Gripper/Grip]);
      SERVER_3 : SERVER_0_1(QI := 1, ID := opc_ua[CREATE_METHOD;/Objects/Turntable/NewPosition]);
      PUBLISH_0 : PUBLISH_1(QI := 1, ID := opc_ua[WRITE;/Objects/Gripper/Gripped]);
      PUBLISH_2 : PUBLISH_1(QI := 1, ID := opc_ua[WRITE;/Objects/Robot/CurrentPosition]);
      PUBLISH_1 : PUBLISH_1(QI := 1, ID := opc_ua[WRITE;/Objects/Gripper/Released]);
      SERVER_1 : SERVER_0(QI := 1, ID := opc_ua[CREATE_METHOD;/Objects/Gripper/Release]);
      SERVER_5 : SERVER_0(QI := 1, ID := opc_ua[CREATE_METHOD;/Objects/Storage/GoOut,1:s=Storage_GoOut]);
      SERVER_4 : SERVER_0(QI := 1, ID := opc_ua[CREATE_METHOD;/Objects/Storage/GoIn,1:s=Storage_GoIn]);
      PUBLISH_4 : PUBLISH_1(QI := 1, ID := opc_ua[WRITE;/Objects/Storage/IsOut]);
      PUBLISH_5 : PUBLISH_1(QI := 1, ID := opc_ua[WRITE;/Objects/Storage/IsIn]);
      SUBSCRIBE_5 : SUBSCRIBE_1(QI := 1, ID := opc_ua[SUBSCRIBE;opc.tcp://localhost:4850#;/Objects/Gripper/Released]);
      CLIENT_4 : CLIENT_0(QI := 1, ID := opc_ua[CALL_METHOD;opc.tcp://localhost:4850#;/Objects/Gripper/Grip]);
      AROBOT_DEMUX : AROBOT_DEMUX;
      HandlingControl : HandlingControl;
      CLIENT_2 : CLIENT_1_0(QI := 1, ID := opc_ua[CALL_METHOD;opc.tcp://localhost:4850#;/Objects/Turntable/NewPosition]);
      SUBSCRIBE_2 : SUBSCRIBE_1(QI := 1, ID := opc_ua[SUBSCRIBE;opc.tcp://localhost:4850#;/Objects/Turntable/CurrentPosition]);
      SUBSCRIBE_4 : SUBSCRIBE_1(QI := 1, ID := opc_ua[SUBSCRIBE;opc.tcp://localhost:4850#;/Objects/Gripper/Gripped]);
      CLIENT_3 : CLIENT_0(QI := 1, ID := opc_ua[CALL_METHOD;opc.tcp://localhost:4850#;/Objects/Storage/GoOut]);
      CLIENT_5 : CLIENT_0(QI := 1, ID := opc_ua[CALL_METHOD;opc.tcp://localhost:4850#;/Objects/Gripper/Release]);
      CLIENT_0 : CLIENT_0(QI := 1, ID := opc_ua[CALL_METHOD;opc.tcp://localhost:4850#;/Objects/Storage/GoIn]);
      SUBSCRIBE_1 : SUBSCRIBE_1(QI := 1, ID := opc_ua[SUBSCRIBE;opc.tcp://localhost:4850#;/Objects/Robot/CurrentPosition]);
      DepotControl : DepotControl;
      CLIENT_1 : CLIENT_1_0(QI := 1, ID := opc_ua[CALL_METHOD;opc.tcp://localhost:4850#;/Objects/Robot/PresetPositionUpd]);
      SUBSCRIBE_0 : SUBSCRIBE_0(QI := 1, ID := opc_ua[SUBSCRIBE;opc.tcp://localhost:4840#]);
      Station1Control : Station1Control;
      SUBSCRIBE_3 : SUBSCRIBE_1(QI := 1, ID := opc_ua[SUBSCRIBE;opc.tcp://localhost:4850#;/Objects/Storage/IsOut]);
      ATURNTABLE_DEMUX : ATURNTABLE_DEMUX;
      SUBSCRIBE_9 : SUBSCRIBE_1(QI := 1, ID := opc_ua[SUBSCRIBE;opc.tcp://localhost:4850#;/Objects/Storage/IsIn]);
      AROBOT_MUX : AROBOT_MUX;
      E_RS_2 : E_RS;
      AGRIPPER_MUX : AGRIPPER_MUX;
      E_RS_3 : E_RS;
      ATURNTABLE_MUX : ATURNTABLE_MUX;
      E_RS : E_RS;
      E_RS_1 : E_RS;
      ASTORAGE_MUX : ASTORAGE_MUX;
      E_SWITCH_2 : E_SWITCH;
      AGRIPPER_DEMUX : AGRIPPER_DEMUX;
      E_SWITCH_3 : E_SWITCH;
      ASTORAGE_DEMUX : ASTORAGE_DEMUX;
      E_SWITCH_1 : E_SWITCH;
      E_SWITCH : E_SWITCH;
    END_FBS
    SUBAPPLICATION Robot
      EVENT_INPUT
        INIT;
      END_EVENT
      EVENT_OUTPUT
        INITO;
      END_EVENT
      SOCKETS
        ARobot : ARobot;
      END_SOCKETS
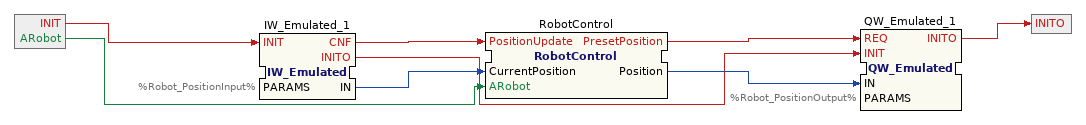
      FBS
        IW_Emulated_1 : IW_Emulated(PARAMS := %Robot_PositionInput%);
        RobotControl : RobotControl;
        QW_Emulated_1 : QW_Emulated(PARAMS := %Robot_PositionOutput%);
      END_FBS
      EVENT_CONNECTIONS
        IW_Emulated_1.CNF TO RobotControl.PositionUpdate;
        RobotControl.PresetPosition TO QW_Emulated_1.REQ;
        IW_Emulated_1.INITO TO QW_Emulated_1.INIT;
        QW_Emulated_1.INITO TO INITO;
        INIT TO IW_Emulated_1.INIT;
      END_CONNECTIONS
      DATA_CONNECTIONS
        IW_Emulated_1.IN TO RobotControl.CurrentPosition;
        RobotControl.Position TO QW_Emulated_1.IN;
      END_CONNECTIONS
      ADAPTER_CONNECTIONS
        ARobot TO RobotControl.ARobot;
      END_CONNECTIONS
    END_SUBAPPLICATION
    SUBAPPLICATION Gripper
      EVENT_INPUT
        INIT;
      END_EVENT
      EVENT_OUTPUT
        INITO;
      END_EVENT
      SOCKETS
        AGripper : AGripper;
      END_SOCKETS
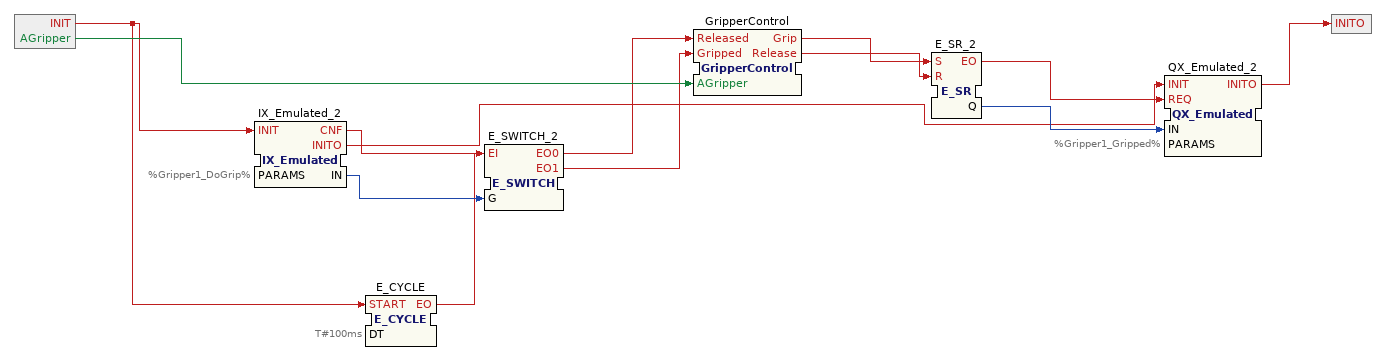
      FBS
        IX_Emulated_2 : IX_Emulated(PARAMS := %Gripper1_DoGrip%);
        E_SWITCH_2 : E_SWITCH;
        GripperControl : GripperControl;
        E_SR_2 : E_SR;
        E_CYCLE : E_CYCLE(DT := T#100ms);
        QX_Emulated_2 : QX_Emulated(PARAMS := %Gripper1_Gripped%);
      END_FBS
      EVENT_CONNECTIONS
        IX_Emulated_2.CNF TO E_SWITCH_2.EI;
        E_SWITCH_2.EO0 TO GripperControl.Released;
        E_SWITCH_2.EO1 TO GripperControl.Gripped;
        GripperControl.Grip TO E_SR_2.S;
        GripperControl.Release TO E_SR_2.R;
        E_CYCLE.EO TO E_SWITCH_2.EI;
        INIT TO E_CYCLE.START;
        INIT TO IX_Emulated_2.INIT;
        IX_Emulated_2.INITO TO QX_Emulated_2.INIT;
        QX_Emulated_2.INITO TO INITO;
        E_SR_2.EO TO QX_Emulated_2.REQ;
      END_CONNECTIONS
      DATA_CONNECTIONS
        IX_Emulated_2.IN TO E_SWITCH_2.G;
        E_SR_2.Q TO QX_Emulated_2.IN;
      END_CONNECTIONS
      ADAPTER_CONNECTIONS
        AGripper TO GripperControl.AGripper;
      END_CONNECTIONS
    END_SUBAPPLICATION
    SUBAPPLICATION Turntable
      EVENT_INPUT
        INIT;
      END_EVENT
      EVENT_OUTPUT
        INITO;
      END_EVENT
      SOCKETS
        ATurntable : ATurntable;
      END_SOCKETS
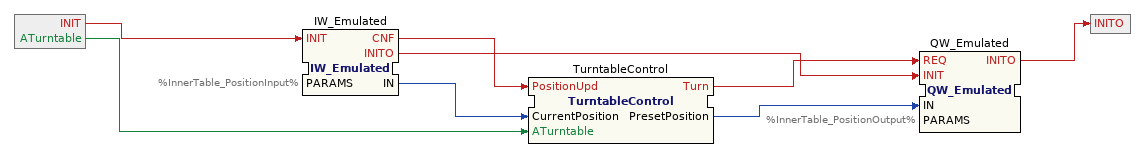
      FBS
        QW_Emulated : QW_Emulated(PARAMS := %InnerTable_PositionOutput%);
        IW_Emulated : IW_Emulated(PARAMS := %InnerTable_PositionInput%);
        TurntableControl : TurntableControl;
      END_FBS
      EVENT_CONNECTIONS
        TurntableControl.Turn TO QW_Emulated.REQ;
        IW_Emulated.CNF TO TurntableControl.PositionUpd;
        IW_Emulated.INITO TO QW_Emulated.INIT;
        INIT TO IW_Emulated.INIT;
        QW_Emulated.INITO TO INITO;
      END_CONNECTIONS
      DATA_CONNECTIONS
        TurntableControl.PresetPosition TO QW_Emulated.IN;
        IW_Emulated.IN TO TurntableControl.CurrentPosition;
      END_CONNECTIONS
      ADAPTER_CONNECTIONS
        ATurntable TO TurntableControl.ATurntable;
      END_CONNECTIONS
    END_SUBAPPLICATION
    SUBAPPLICATION Storage
      EVENT_INPUT
        INIT;
      END_EVENT
      EVENT_OUTPUT
        INITO;
      END_EVENT
      SOCKETS
        AStorage : AStorage;
      END_SOCKETS
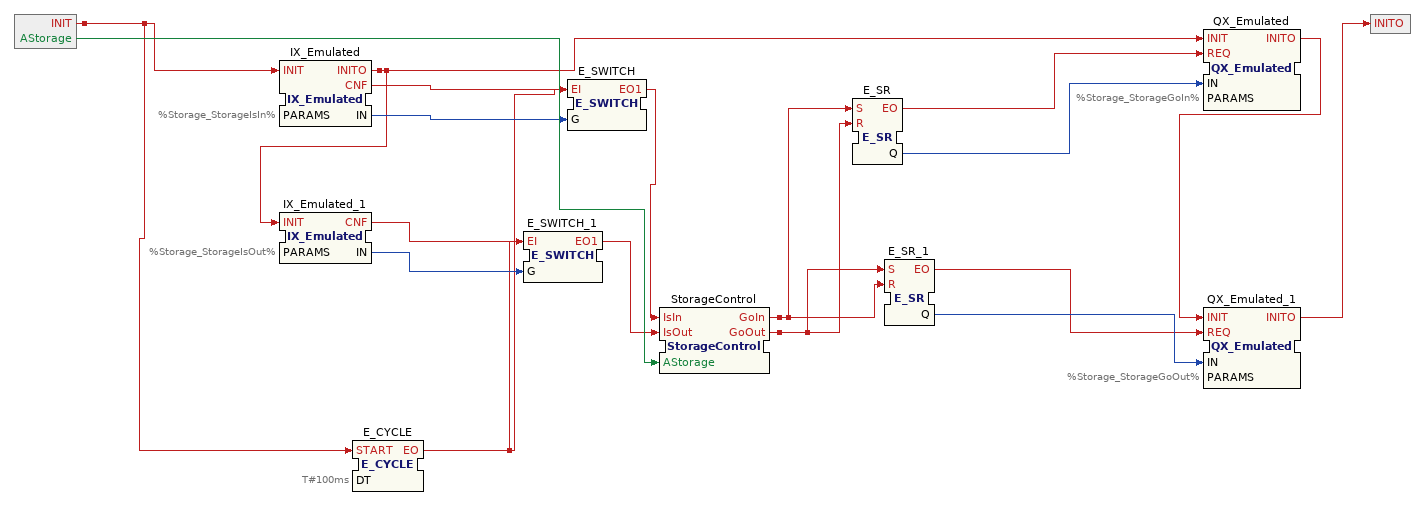
      FBS
        IX_Emulated : IX_Emulated(PARAMS := %Storage_StorageIsIn%);
        E_SWITCH : E_SWITCH;
        E_SR : E_SR;
        E_SR_1 : E_SR;
        StorageControl : StorageControl;
        E_SWITCH_1 : E_SWITCH;
        IX_Emulated_1 : IX_Emulated(PARAMS := %Storage_StorageIsOut%);
        E_CYCLE : E_CYCLE(DT := T#100ms);
        QX_Emulated_1 : QX_Emulated(PARAMS := %Storage_StorageGoOut%);
        QX_Emulated : QX_Emulated(PARAMS := %Storage_StorageGoIn%);
      END_FBS
      EVENT_CONNECTIONS
        IX_Emulated.INITO TO IX_Emulated_1.INIT;
        IX_Emulated.CNF TO E_SWITCH.EI;
        E_SWITCH.EO1 TO StorageControl.IsIn;
        StorageControl.GoIn TO E_SR.S;
        StorageControl.GoOut TO E_SR.R;
        StorageControl.GoOut TO E_SR_1.S;
        StorageControl.GoIn TO E_SR_1.R;
        E_SWITCH_1.EO1 TO StorageControl.IsOut;
        IX_Emulated_1.CNF TO E_SWITCH_1.EI;
        INIT TO IX_Emulated.INIT;
        INIT TO E_CYCLE.START;
        QX_Emulated_1.INITO TO INITO;
        IX_Emulated.INITO TO QX_Emulated.INIT;
        QX_Emulated.INITO TO QX_Emulated_1.INIT;
        E_SR.EO TO QX_Emulated.REQ;
        E_SR_1.EO TO QX_Emulated_1.REQ;
        E_CYCLE.EO TO E_SWITCH.EI;
        E_CYCLE.EO TO E_SWITCH_1.EI;
      END_CONNECTIONS
      DATA_CONNECTIONS
        IX_Emulated.IN TO E_SWITCH.G;
        IX_Emulated_1.IN TO E_SWITCH_1.G;
        E_SR.Q TO QX_Emulated.IN;
        E_SR_1.Q TO QX_Emulated_1.IN;
      END_CONNECTIONS
      ADAPTER_CONNECTIONS
        AStorage TO StorageControl.AStorage;
      END_CONNECTIONS
    END_SUBAPPLICATION
    EVENT_CONNECTIONS
      SERVER_1.IND TO SERVER_1.RSP;
      SERVER_1.INITO TO PUBLISH_0.INIT;
      SERVER_2.IND TO SERVER_2.RSP;
      SERVER_2.INITO TO PUBLISH_2.INIT;
      PUBLISH_0.INITO TO PUBLISH_1.INIT;
      SERVER_0.INITO TO SERVER_1.INIT;
      SERVER_3.IND TO SERVER_3.RSP;
      SERVER_0.IND TO SERVER_0.RSP;
      SERVER_3.INITO TO PUBLISH_3.INIT;
      SERVER_5.IND TO SERVER_5.RSP;
      PUBLISH_5.INITO TO PUBLISH_4.INIT;
      SERVER_4.INITO TO SERVER_5.INIT;
      SERVER_5.INITO TO PUBLISH_5.INIT;
      SERVER_4.IND TO SERVER_4.RSP;
      SUBSCRIBE_2.IND TO ATURNTABLE_DEMUX.PositionUpd;
      CLIENT_4.INITO TO CLIENT_5.INIT;
      CLIENT_0.INITO TO CLIENT_3.INIT;
      CLIENT_3.INITO TO SUBSCRIBE_2.INIT;
      SUBSCRIBE_2.INITO TO SUBSCRIBE_4.INIT;
      SUBSCRIBE_2.INITO TO CLIENT_2.INIT;
      SUBSCRIBE_5.INITO TO SUBSCRIBE_1.INIT;
      SUBSCRIBE_1.INITO TO CLIENT_1.INIT;
      SUBSCRIBE_4.INITO TO SUBSCRIBE_5.INIT;
      SUBSCRIBE_3.INITO TO CLIENT_0.INIT;
      ATURNTABLE_DEMUX.NewPosition TO CLIENT_2.REQ;
      SUBSCRIBE_9.INITO TO SUBSCRIBE_3.INIT;
      AROBOT_DEMUX.PresetPositionUpd TO CLIENT_1.REQ;
      SUBSCRIBE_5.INITO TO CLIENT_4.INIT;
      SUBSCRIBE_1.IND TO AROBOT_DEMUX.PositionUpdate;
      CLIENT_0.INITO TO SERVER_4.INIT;
      Robot.INITO TO SERVER_2.INIT;
      AROBOT_MUX.PositionUpdate TO PUBLISH_2.REQ;
      SERVER_2.IND TO AROBOT_MUX.PresetPositionUpd;
      E_RS_3.EO TO PUBLISH_1.REQ;
      Gripper.INITO TO SERVER_0.INIT;
      Gripper.INITO TO Robot.INIT;
      SERVER_1.IND TO AGRIPPER_MUX.Release;
      SERVER_0.IND TO AGRIPPER_MUX.Grip;
      E_RS_2.EO TO PUBLISH_0.REQ;
      AGRIPPER_MUX.Released TO E_RS_2.R;
      AGRIPPER_MUX.Gripped TO E_RS_2.S;
      AGRIPPER_MUX.Gripped TO E_RS_3.R;
      AGRIPPER_MUX.Released TO E_RS_3.S;
      Turntable.INITO TO Gripper.INIT;
      Turntable.INITO TO SERVER_3.INIT;
      ATURNTABLE_MUX.PositionUpd TO PUBLISH_3.REQ;
      SERVER_3.IND TO ATURNTABLE_MUX.NewPosition;
      SERVER_5.IND TO ASTORAGE_MUX.GoOut;
      SERVER_4.IND TO ASTORAGE_MUX.GoIn;
      Storage.INITO TO Turntable.INIT;
      SERVER_5.INITO TO Storage.INIT;
      E_RS_1.EO TO PUBLISH_5.REQ;
      E_RS.EO TO PUBLISH_4.REQ;
      ASTORAGE_MUX.IsIn TO E_RS.R;
      ASTORAGE_MUX.IsOut TO E_RS.S;
      ASTORAGE_MUX.IsOut TO E_RS_1.R;
      ASTORAGE_MUX.IsIn TO E_RS_1.S;
      SUBSCRIBE_5.IND TO E_SWITCH_3.EI;
      AGRIPPER_DEMUX.Release TO CLIENT_5.REQ;
      AGRIPPER_DEMUX.Grip TO CLIENT_4.REQ;
      SUBSCRIBE_4.IND TO E_SWITCH_2.EI;
      AGRIPPER_DEMUX.Grip TO E_SWITCH_2.EI;
      E_SWITCH_2.EO1 TO AGRIPPER_DEMUX.Gripped;
      E_SWITCH_3.EO1 TO AGRIPPER_DEMUX.Released;
      AGRIPPER_DEMUX.Release TO E_SWITCH_3.EI;
      SUBSCRIBE_3.IND TO E_SWITCH.EI;
      SUBSCRIBE_9.IND TO E_SWITCH_1.EI;
      ASTORAGE_DEMUX.GoOut TO CLIENT_3.REQ;
      ASTORAGE_DEMUX.GoIn TO CLIENT_0.REQ;
      E_SWITCH_1.EO1 TO ASTORAGE_DEMUX.IsIn;
      E_SWITCH.EO1 TO ASTORAGE_DEMUX.IsOut;
      ASTORAGE_DEMUX.GoIn TO E_SWITCH_1.EI;
      ASTORAGE_DEMUX.GoOut TO E_SWITCH.EI;
    END_CONNECTIONS
    DATA_CONNECTIONS
      SUBSCRIBE_2.RD_1 TO ATURNTABLE_DEMUX.CurrentPosition;
      ATURNTABLE_DEMUX.Position TO CLIENT_2.SD_1;
      SUBSCRIBE_1.RD_1 TO AROBOT_DEMUX.CurrentPosition;
      AROBOT_DEMUX.PresetPosition TO CLIENT_1.SD_1;
      AROBOT_MUX.CurrentPosition TO PUBLISH_2.SD_1;
      SERVER_2.RD_1 TO AROBOT_MUX.PresetPosition;
      E_RS_3.Q TO PUBLISH_1.SD_1;
      E_RS_2.Q TO PUBLISH_0.SD_1;
      ATURNTABLE_MUX.CurrentPosition TO PUBLISH_3.SD_1;
      SERVER_3.RD_1 TO ATURNTABLE_MUX.Position;
      E_RS_1.Q TO PUBLISH_5.SD_1;
      E_RS.Q TO PUBLISH_4.SD_1;
      SUBSCRIBE_5.RD_1 TO E_SWITCH_3.G;
      SUBSCRIBE_4.RD_1 TO E_SWITCH_2.G;
      SUBSCRIBE_3.RD_1 TO E_SWITCH.G;
      SUBSCRIBE_9.RD_1 TO E_SWITCH_1.G;
    END_CONNECTIONS
    ADAPTER_CONNECTIONS
      Station1Control.ADepot TO DepotControl.ADepot;
      Station1Control.AHandling TO HandlingControl.AHandling;
      HandlingControl.ARobot TO AROBOT_DEMUX.ARobot;
      DepotControl.ATurntable TO ATURNTABLE_DEMUX.ATurntable;
      AROBOT_MUX.ARobot TO Robot.ARobot;
      AGRIPPER_MUX.AGripper TO Gripper.AGripper;
      ATURNTABLE_MUX.ATurntable TO Turntable.ATurntable;
      ASTORAGE_MUX.AStorage TO Storage.AStorage;
      HandlingControl.AGripper TO AGRIPPER_DEMUX.AGripper;
      DepotControl.AStorage TO ASTORAGE_DEMUX.AStorage;
    END_CONNECTIONS
  END_APPLICATION
  APPLICATION VDMA_Station1_SkillbasedControl_Distributed_SingleDevice
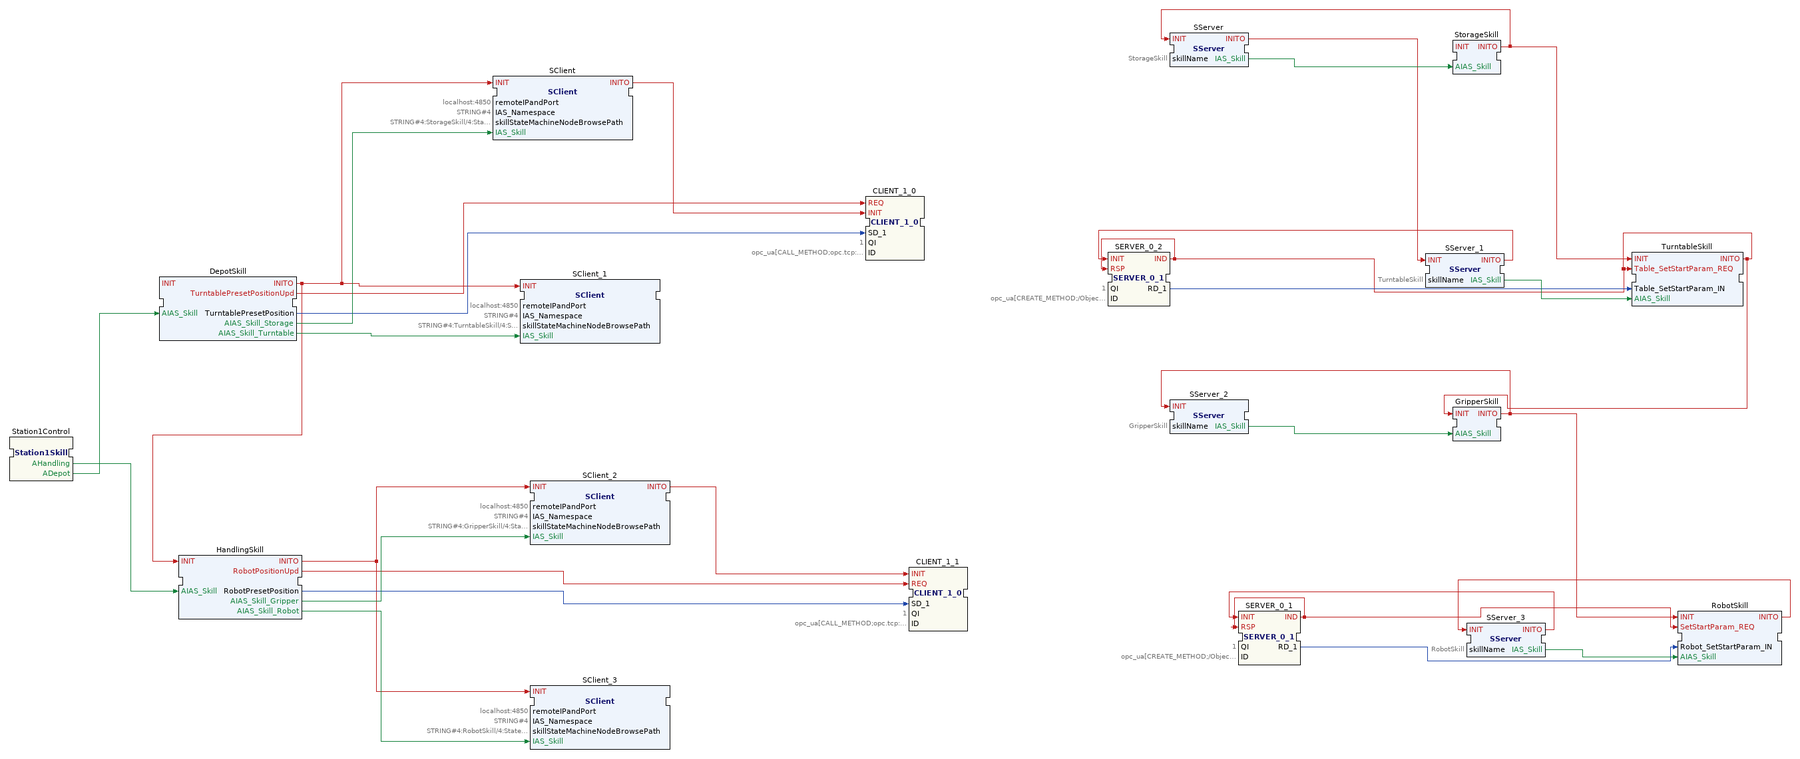
    FBS
      Station1Control : Station1Skill;
      SERVER_0_1 : SERVER_0_1(QI := 1, ID := opc_ua[CREATE_METHOD;/Objects/4:RobotSkill/4:SetStartParams]);
      SERVER_0_2 : SERVER_0_1(QI := 1, ID := opc_ua[CREATE_METHOD;/Objects/4:TurntableSkill/4:SetStartParams]);
      CLIENT_1_0 : CLIENT_1_0(QI := 1, ID := opc_ua[CALL_METHOD;opc.tcp://localhost:4850#;/Objects/4:TurntableSkill/4:SetStartParams]);
      CLIENT_1_1 : CLIENT_1_0(QI := 1, ID := opc_ua[CALL_METHOD;opc.tcp://localhost:4850#;/Objects/4:RobotSkill/4:SetStartParams]);
    END_FBS
    SUBAPPS
      SServer : SServer(skillName := StorageSkill);
      SServer_1 : SServer(skillName := TurntableSkill);
      SServer_2 : SServer(skillName := GripperSkill);
      SServer_3 : SServer(skillName := RobotSkill);
      SClient_1 : SClient(remoteIPandPort := localhost:4850, IAS_Namespace := STRING#4, skillStateMachineNodeBrowsePath := STRING#4:TurntableSkill/4:StateMachine/);
      SClient_2 : SClient(remoteIPandPort := localhost:4850, IAS_Namespace := STRING#4, skillStateMachineNodeBrowsePath := STRING#4:GripperSkill/4:StateMachine/);
      SClient_3 : SClient(remoteIPandPort := localhost:4850, IAS_Namespace := STRING#4, skillStateMachineNodeBrowsePath := STRING#4:RobotSkill/4:StateMachine/);
      SClient : SClient(remoteIPandPort := localhost:4850, IAS_Namespace := STRING#4, skillStateMachineNodeBrowsePath := STRING#4:StorageSkill/4:StateMachine/);
    END_SUBAPPS
    SUBAPPLICATION StorageSkill
      EVENT_INPUT
        INIT;
      END_EVENT
      EVENT_OUTPUT
        INITO;
      END_EVENT
      SOCKETS
        AIAS_Skill : IAS_Skill;
      END_SOCKETS
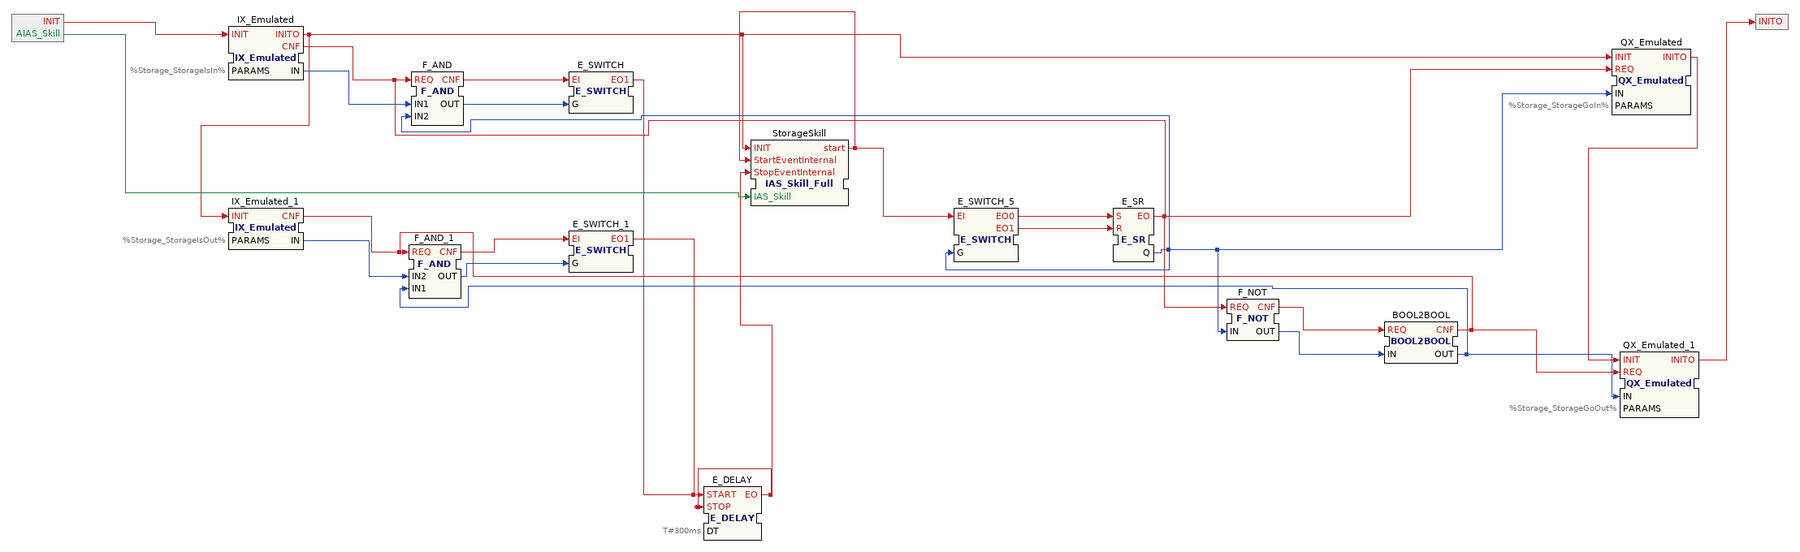
      FBS
        E_SWITCH_5 : E_SWITCH;
        IX_Emulated : IX_Emulated(PARAMS := %Storage_StorageIsIn%);
        F_NOT : F_NOT;
        IX_Emulated_1 : IX_Emulated(PARAMS := %Storage_StorageIsOut%);
        E_SWITCH : E_SWITCH;
        E_SWITCH_1 : E_SWITCH;
        StorageSkill : IAS_Skill_Full;
        F_AND : F_AND;
        BOOL2BOOL : BOOL2BOOL;
        F_AND_1 : F_AND;
        E_SR : E_SR;
        QX_Emulated : QX_Emulated(PARAMS := %Storage_StorageGoIn%);
        QX_Emulated_1 : QX_Emulated(PARAMS := %Storage_StorageGoOut%);
        E_DELAY : E_DELAY(DT := T#300ms);
      END_FBS
      EVENT_CONNECTIONS
        StorageSkill.start TO E_SWITCH_5.EI;
        E_SWITCH_5.EO0 TO E_SR.S;
        E_SWITCH_5.EO1 TO E_SR.R;
        IX_Emulated.INITO TO IX_Emulated_1.INIT;
        IX_Emulated.INITO TO StorageSkill.INIT;
        IX_Emulated.CNF TO F_AND.REQ;
        E_SR.EO TO F_NOT.REQ;
        F_NOT.CNF TO BOOL2BOOL.REQ;
        IX_Emulated_1.CNF TO F_AND_1.REQ;
        F_AND.CNF TO E_SWITCH.EI;
        F_AND_1.CNF TO E_SWITCH_1.EI;
        StorageSkill.start TO StorageSkill.StartEventInternal;
        E_SR.EO TO F_AND.REQ;
        BOOL2BOOL.CNF TO F_AND_1.REQ;
        INIT TO IX_Emulated.INIT;
        IX_Emulated.INITO TO QX_Emulated.INIT;
        QX_Emulated.INITO TO QX_Emulated_1.INIT;
        QX_Emulated_1.INITO TO INITO;
        BOOL2BOOL.CNF TO QX_Emulated_1.REQ;
        E_SR.EO TO QX_Emulated.REQ;
        E_SWITCH.EO1 TO E_DELAY.START;
        E_SWITCH_1.EO1 TO E_DELAY.START;
        E_DELAY.EO TO StorageSkill.StopEventInternal;
        E_DELAY.EO TO E_DELAY.STOP;
      END_CONNECTIONS
      DATA_CONNECTIONS
        E_SR.Q TO E_SWITCH_5.G;
        IX_Emulated.IN TO F_AND.IN1;
        E_SR.Q TO F_NOT.IN;
        F_NOT.OUT TO BOOL2BOOL.IN;
        IX_Emulated_1.IN TO F_AND_1.IN2;
        F_AND.OUT TO E_SWITCH.G;
        F_AND_1.OUT TO E_SWITCH_1.G;
        E_SR.Q TO F_AND.IN2;
        BOOL2BOOL.OUT TO F_AND_1.IN1;
        BOOL2BOOL.OUT TO QX_Emulated_1.IN;
        E_SR.Q TO QX_Emulated.IN;
      END_CONNECTIONS
      ADAPTER_CONNECTIONS
        AIAS_Skill TO StorageSkill.IAS_Skill;
      END_CONNECTIONS
    END_SUBAPPLICATION
    SUBAPPLICATION TurntableSkill
      EVENT_INPUT
        INIT;
        Table_SetStartParam_REQ;
      END_EVENT
      EVENT_OUTPUT
        INITO;
      END_EVENT
      VAR_INPUT
        Table_SetStartParam_IN : WORD;
      END_VAR
      SOCKETS
        AIAS_Skill : IAS_Skill;
      END_SOCKETS
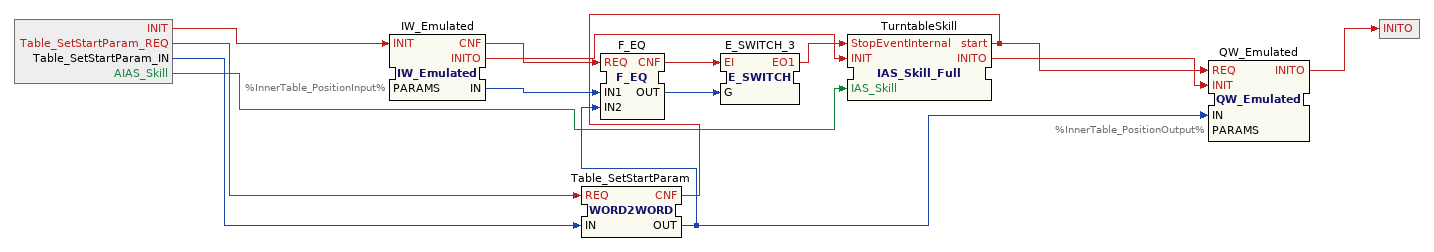
      FBS
        F_EQ : F_EQ;
        E_SWITCH_3 : E_SWITCH;
        Table_SetStartParam : WORD2WORD;
        QW_Emulated : QW_Emulated(PARAMS := %InnerTable_PositionOutput%);
        TurntableSkill : IAS_Skill_Full;
        IW_Emulated : IW_Emulated(PARAMS := %InnerTable_PositionInput%);
      END_FBS
      EVENT_CONNECTIONS
        IW_Emulated.CNF TO F_EQ.REQ;
        TurntableSkill.start TO F_EQ.REQ;
        Table_SetStartParam.CNF TO F_EQ.REQ;
        F_EQ.CNF TO E_SWITCH_3.EI;
        E_SWITCH_3.EO1 TO TurntableSkill.StopEventInternal;
        TurntableSkill.start TO QW_Emulated.REQ;
        Table_SetStartParam_REQ TO Table_SetStartParam.REQ;
        INIT TO IW_Emulated.INIT;
        IW_Emulated.INITO TO TurntableSkill.INIT;
        TurntableSkill.INITO TO QW_Emulated.INIT;
        QW_Emulated.INITO TO INITO;
      END_CONNECTIONS
      DATA_CONNECTIONS
        IW_Emulated.IN TO F_EQ.IN1;
        Table_SetStartParam.OUT TO F_EQ.IN2;
        F_EQ.OUT TO E_SWITCH_3.G;
        Table_SetStartParam.OUT TO QW_Emulated.IN;
        Table_SetStartParam_IN TO Table_SetStartParam.IN;
      END_CONNECTIONS
      ADAPTER_CONNECTIONS
        AIAS_Skill TO TurntableSkill.IAS_Skill;
      END_CONNECTIONS
    END_SUBAPPLICATION
    SUBAPPLICATION DepotSkill
      EVENT_INPUT
        INIT;
      END_EVENT
      EVENT_OUTPUT
        INITO;
        TurntablePresetPositionUpd;
      END_EVENT
      VAR_OUTPUT
        TurntablePresetPosition : WORD;
      END_VAR
      SOCKETS
        AIAS_Skill : IAS_Skill;
      END_SOCKETS
      PLUGS
        AIAS_Skill_Storage : IAS_Skill;
        AIAS_Skill_Turntable : IAS_Skill;
      END_PLUGS
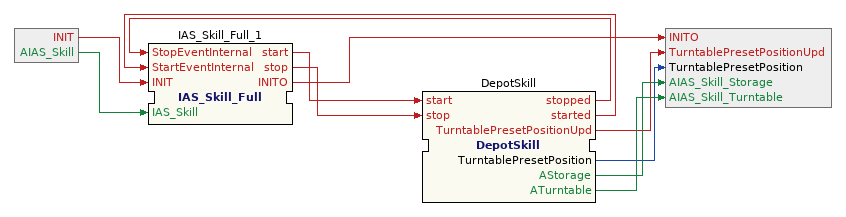
      FBS
        IAS_Skill_Full_1 : IAS_Skill_Full;
        DepotSkill : DepotSkill;
      END_FBS
      EVENT_CONNECTIONS
        DepotSkill.stopped TO IAS_Skill_Full_1.StopEventInternal;
        DepotSkill.started TO IAS_Skill_Full_1.StartEventInternal;
        IAS_Skill_Full_1.start TO DepotSkill.start;
        IAS_Skill_Full_1.stop TO DepotSkill.stop;
        DepotSkill.TurntablePresetPositionUpd TO TurntablePresetPositionUpd;
        INIT TO IAS_Skill_Full_1.INIT;
        IAS_Skill_Full_1.INITO TO INITO;
      END_CONNECTIONS
      DATA_CONNECTIONS
        DepotSkill.TurntablePresetPosition TO TurntablePresetPosition;
      END_CONNECTIONS
      ADAPTER_CONNECTIONS
        AIAS_Skill TO IAS_Skill_Full_1.IAS_Skill;
        DepotSkill.AStorage TO AIAS_Skill_Storage;
        DepotSkill.ATurntable TO AIAS_Skill_Turntable;
      END_CONNECTIONS
    END_SUBAPPLICATION
    SUBAPPLICATION GripperSkill
      EVENT_INPUT
        INIT;
      END_EVENT
      EVENT_OUTPUT
        INITO;
      END_EVENT
      SOCKETS
        AIAS_Skill : IAS_Skill;
      END_SOCKETS
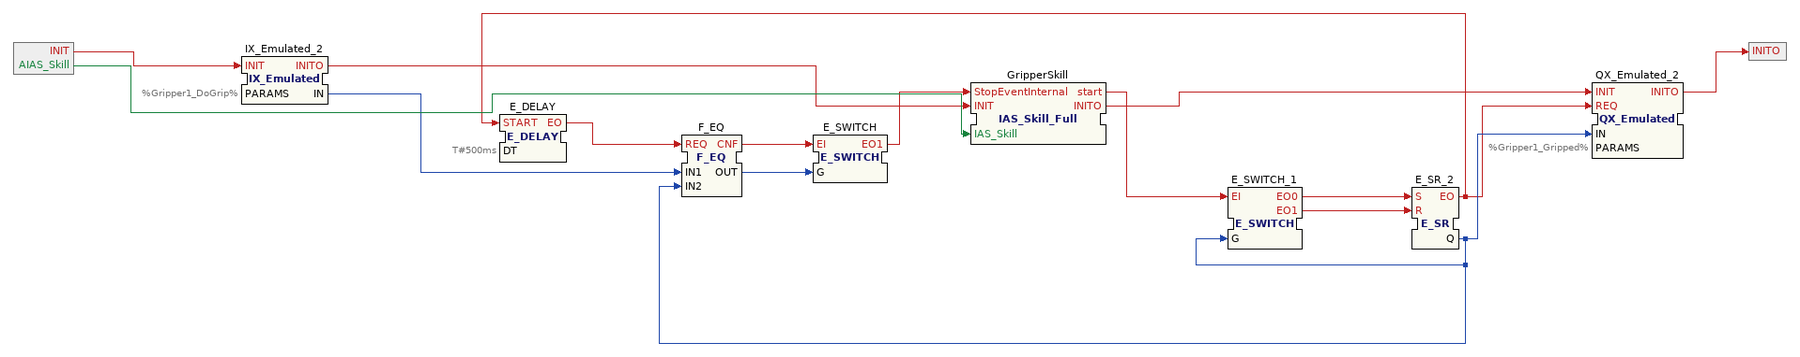
      FBS
        GripperSkill : IAS_Skill_Full;
        F_EQ : F_EQ;
        E_SWITCH_1 : E_SWITCH;
        IX_Emulated_2 : IX_Emulated(PARAMS := %Gripper1_DoGrip%);
        E_DELAY : E_DELAY(DT := T#500ms);
        E_SWITCH : E_SWITCH;
        E_SR_2 : E_SR;
        QX_Emulated_2 : QX_Emulated(PARAMS := %Gripper1_Gripped%);
      END_FBS
      EVENT_CONNECTIONS
        E_SWITCH.EO1 TO GripperSkill.StopEventInternal;
        GripperSkill.start TO E_SWITCH_1.EI;
        E_DELAY.EO TO F_EQ.REQ;
        F_EQ.CNF TO E_SWITCH.EI;
        E_SWITCH_1.EO0 TO E_SR_2.S;
        E_SWITCH_1.EO1 TO E_SR_2.R;
        E_SR_2.EO TO E_DELAY.START;
        INIT TO IX_Emulated_2.INIT;
        IX_Emulated_2.INITO TO GripperSkill.INIT;
        GripperSkill.INITO TO QX_Emulated_2.INIT;
        QX_Emulated_2.INITO TO INITO;
        E_SR_2.EO TO QX_Emulated_2.REQ;
      END_CONNECTIONS
      DATA_CONNECTIONS
        IX_Emulated_2.IN TO F_EQ.IN1;
        E_SR_2.Q TO F_EQ.IN2;
        F_EQ.OUT TO E_SWITCH.G;
        E_SR_2.Q TO E_SWITCH_1.G;
        E_SR_2.Q TO QX_Emulated_2.IN;
      END_CONNECTIONS
      ADAPTER_CONNECTIONS
        AIAS_Skill TO GripperSkill.IAS_Skill;
      END_CONNECTIONS
    END_SUBAPPLICATION
    SUBAPPLICATION RobotSkill
      EVENT_INPUT
        INIT;
        SetStartParam_REQ;
      END_EVENT
      EVENT_OUTPUT
        INITO;
      END_EVENT
      VAR_INPUT
        Robot_SetStartParam_IN : WORD;
      END_VAR
      SOCKETS
        AIAS_Skill : IAS_Skill;
      END_SOCKETS
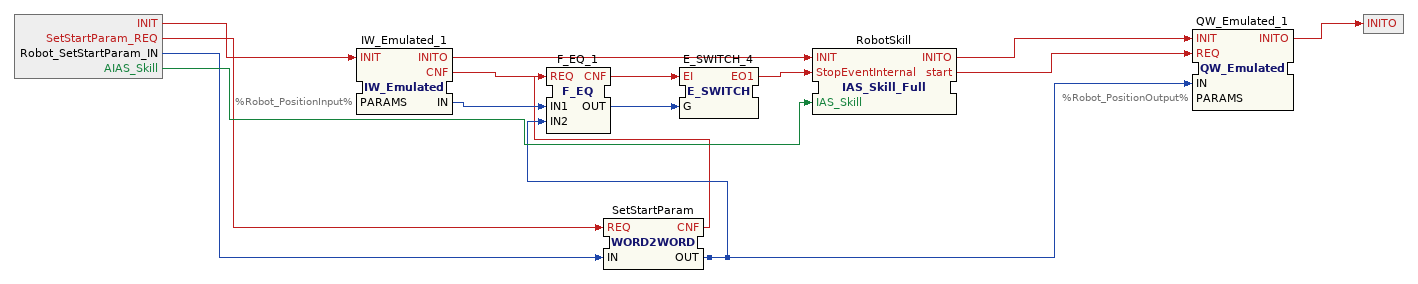
      FBS
        RobotSkill : IAS_Skill_Full;
        IW_Emulated_1 : IW_Emulated(PARAMS := %Robot_PositionInput%);
        E_SWITCH_4 : E_SWITCH;
        F_EQ_1 : F_EQ;
        QW_Emulated_1 : QW_Emulated(PARAMS := %Robot_PositionOutput%);
        SetStartParam : WORD2WORD;
      END_FBS
      EVENT_CONNECTIONS
        IW_Emulated_1.INITO TO RobotSkill.INIT;
        E_SWITCH_4.EO1 TO RobotSkill.StopEventInternal;
        RobotSkill.INITO TO QW_Emulated_1.INIT;
        RobotSkill.start TO QW_Emulated_1.REQ;
        IW_Emulated_1.CNF TO F_EQ_1.REQ;
        F_EQ_1.CNF TO E_SWITCH_4.EI;
        SetStartParam.CNF TO F_EQ_1.REQ;
        INIT TO IW_Emulated_1.INIT;
        SetStartParam_REQ TO SetStartParam.REQ;
        QW_Emulated_1.INITO TO INITO;
      END_CONNECTIONS
      DATA_CONNECTIONS
        IW_Emulated_1.IN TO F_EQ_1.IN1;
        F_EQ_1.OUT TO E_SWITCH_4.G;
        SetStartParam.OUT TO F_EQ_1.IN2;
        SetStartParam.OUT TO QW_Emulated_1.IN;
        Robot_SetStartParam_IN TO SetStartParam.IN;
      END_CONNECTIONS
      ADAPTER_CONNECTIONS
        AIAS_Skill TO RobotSkill.IAS_Skill;
      END_CONNECTIONS
    END_SUBAPPLICATION
    SUBAPPLICATION HandlingSkill
      EVENT_INPUT
        INIT;
      END_EVENT
      EVENT_OUTPUT
        INITO;
        RobotPositionUpd;
      END_EVENT
      VAR_OUTPUT
        RobotPresetPosition : WORD;
      END_VAR
      SOCKETS
        AIAS_Skill : IAS_Skill;
      END_SOCKETS
      PLUGS
        AIAS_Skill_Gripper : IAS_Skill;
        AIAS_Skill_Robot : IAS_Skill;
      END_PLUGS
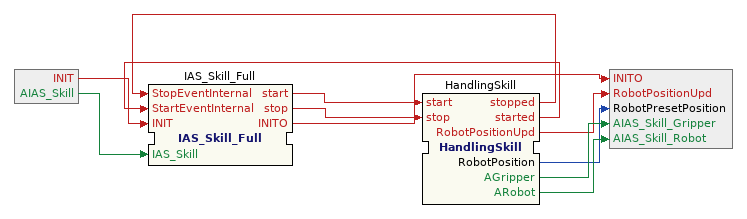
      FBS
        IAS_Skill_Full : IAS_Skill_Full;
        HandlingSkill : HandlingSkill;
      END_FBS
      EVENT_CONNECTIONS
        HandlingSkill.stopped TO IAS_Skill_Full.StopEventInternal;
        HandlingSkill.started TO IAS_Skill_Full.StartEventInternal;
        IAS_Skill_Full.start TO HandlingSkill.start;
        IAS_Skill_Full.stop TO HandlingSkill.stop;
        HandlingSkill.RobotPositionUpd TO RobotPositionUpd;
        INIT TO IAS_Skill_Full.INIT;
        IAS_Skill_Full.INITO TO INITO;
      END_CONNECTIONS
      DATA_CONNECTIONS
        HandlingSkill.RobotPosition TO RobotPresetPosition;
      END_CONNECTIONS
      ADAPTER_CONNECTIONS
        AIAS_Skill TO IAS_Skill_Full.IAS_Skill;
        HandlingSkill.AGripper TO AIAS_Skill_Gripper;
        HandlingSkill.ARobot TO AIAS_Skill_Robot;
      END_CONNECTIONS
    END_SUBAPPLICATION
    EVENT_CONNECTIONS
      DepotSkill.INITO TO SClient_1.INIT;
      TurntableSkill.INITO TO TurntableSkill.Table_SetStartParam_REQ;
      GripperSkill.INITO TO SServer_2.INIT;
      HandlingSkill.INITO TO SClient_3.INIT;
      DepotSkill.INITO TO HandlingSkill.INIT;
      StorageSkill.INITO TO SServer.INIT;
      HandlingSkill.INITO TO SClient_2.INIT;
      StorageSkill.INITO TO TurntableSkill.INIT;
      TurntableSkill.INITO TO GripperSkill.INIT;
      GripperSkill.INITO TO RobotSkill.INIT;
      DepotSkill.INITO TO SClient.INIT;
      SERVER_0_1.IND TO RobotSkill.SetStartParam_REQ;
      SERVER_0_2.IND TO TurntableSkill.Table_SetStartParam_REQ;
      DepotSkill.TurntablePresetPositionUpd TO CLIENT_1_0.REQ;
      SClient.INITO TO CLIENT_1_0.INIT;
      SClient_2.INITO TO CLIENT_1_1.INIT;
      HandlingSkill.RobotPositionUpd TO CLIENT_1_1.REQ;
      SServer.INITO TO SServer_1.INIT;
      RobotSkill.INITO TO SServer_3.INIT;
      SServer_3.INITO TO SERVER_0_1.INIT;
      SServer_1.INITO TO SERVER_0_2.INIT;
      SERVER_0_2.IND TO SERVER_0_2.RSP;
      SERVER_0_1.IND TO SERVER_0_1.RSP;
    END_CONNECTIONS
    DATA_CONNECTIONS
      SERVER_0_1.RD_1 TO RobotSkill.Robot_SetStartParam_IN;
      SERVER_0_2.RD_1 TO TurntableSkill.Table_SetStartParam_IN;
      DepotSkill.TurntablePresetPosition TO CLIENT_1_0.SD_1;
      HandlingSkill.RobotPresetPosition TO CLIENT_1_1.SD_1;
    END_CONNECTIONS
    ADAPTER_CONNECTIONS
      SServer_1.IAS_Skill TO TurntableSkill.AIAS_Skill;
      DepotSkill.AIAS_Skill_Turntable TO SClient_1.IAS_Skill;
      SServer_2.IAS_Skill TO GripperSkill.AIAS_Skill;
      Station1Control.AHandling TO HandlingSkill.AIAS_Skill;
      HandlingSkill.AIAS_Skill_Gripper TO SClient_2.IAS_Skill;
      HandlingSkill.AIAS_Skill_Robot TO SClient_3.IAS_Skill;
      SServer.IAS_Skill TO StorageSkill.AIAS_Skill;
      SServer_3.IAS_Skill TO RobotSkill.AIAS_Skill;
      Station1Control.ADepot TO DepotSkill.AIAS_Skill;
      DepotSkill.AIAS_Skill_Storage TO SClient.IAS_Skill;
    END_CONNECTIONS
  END_APPLICATION
  APPLICATION VDMA_Station1_CodeGenDistributed
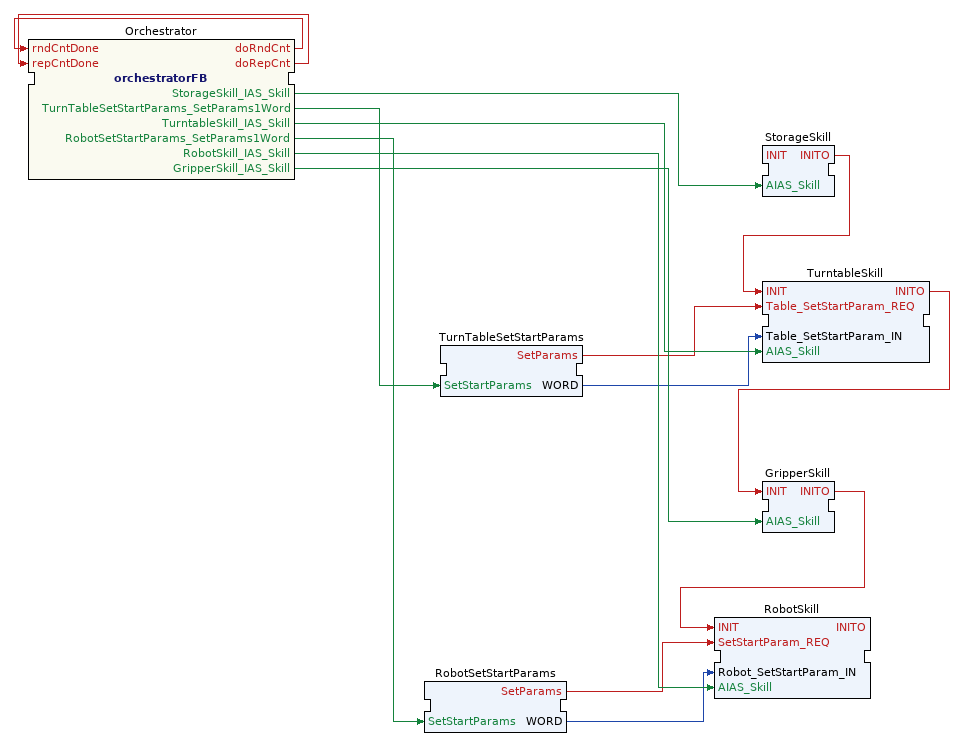
    FBS
      Orchestrator : orchestratorFB;
    END_FBS
    SUBAPPLICATION TurnTableSetStartParams
      EVENT_OUTPUT
        SetParams;
      END_EVENT
      VAR_OUTPUT
        WORD : WORD;
      END_VAR
      SOCKETS
        SetStartParams : SetParams1Word;
      END_SOCKETS
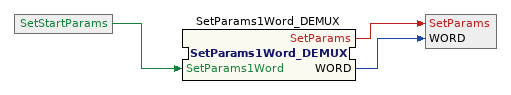
      FBS
        SetParams1Word_DEMUX : SetParams1Word_DEMUX;
      END_FBS
      EVENT_CONNECTIONS
        SetParams1Word_DEMUX.SetParams TO SetParams;
      END_CONNECTIONS
      DATA_CONNECTIONS
        SetParams1Word_DEMUX.WORD TO WORD;
      END_CONNECTIONS
      ADAPTER_CONNECTIONS
        SetStartParams TO SetParams1Word_DEMUX.SetParams1Word;
      END_CONNECTIONS
    END_SUBAPPLICATION
    SUBAPPLICATION RobotSetStartParams
      EVENT_OUTPUT
        SetParams;
      END_EVENT
      VAR_OUTPUT
        WORD : WORD;
      END_VAR
      SOCKETS
        SetStartParams : SetParams1Word;
      END_SOCKETS
